	IF Cylinder.List.fbUpCV_FeedInPress1.xError THEN
		Cylinder.List.fbUpCV_FeedInPress1.M_Reset();
	END_IF
	IF Cylinder.List.fbUpCV_FeedInPress2.xError THEN
		Cylinder.List.fbUpCV_FeedInPress2.M_Reset();
	END_IF
	IF Cylinder.List.fbUpCV_DiameterPress.xError THEN
		Cylinder.List.fbUpCV_DiameterPress.M_Reset();
	END_IF
	IF Cylinder.List.fbUpCV_CamaraPress1.xError THEN
		Cylinder.List.fbUpCV_CamaraPress1.M_Reset();
	END_IF
	IF Cylinder.List.fbUpCV_CamaraPress2.xError THEN
		Cylinder.List.fbUpCV_CamaraPress2.M_Reset();
	END_IF
	IF Cylinder.List.fbUpCV_CamaraPress3.xError THEN
		Cylinder.List.fbUpCV_CamaraPress3.M_Reset();
	END_IF
	IF Cylinder.List.fbUpCV_CamaraPress4.xError THEN
		Cylinder.List.fbUpCV_CamaraPress4.M_Reset();
	END_IF
	IF Cylinder.List.fbUpCV_Block1.xError THEN
		Cylinder.List.fbUpCV_Block1.M_Reset();
	END_IF
	IF Cylinder.List.fbUpCV_Block2.xError THEN
		Cylinder.List.fbUpCV_Block2.M_Reset();
	END_IF
	IF Cylinder.List.fbUpCV_Block3.xError THEN
		Cylinder.List.fbUpCV_Block3.M_Reset();
	END_IF
	IF Cylinder.List.fbUpCV_DiameterHoriz.xError THEN
		Cylinder.List.fbUpCV_DiameterHoriz.M_Reset();
	END_IF
	IF Cylinder.List.fbUpCV_DiameterVert.xError THEN
		Cylinder.List.fbUpCV_DiameterVert.M_Reset();
	END_IF
	IF Cylinder.List.fbUpCV_DiameterClamp.xError THEN
		Cylinder.List.fbUpCV_DiameterClamp.M_Reset();
	END_IF
	IF Cylinder.List.fbStackPush.xError THEN
		Cylinder.List.fbStackPush.M_Reset();
	END_IF
	IF Cylinder.List.fbPullOutCV_AsidePress1.xError THEN
		Cylinder.List.fbPullOutCV_AsidePress1.M_Reset();
	END_IF
	IF Cylinder.List.fbPullOutCV_AsidePress2.xError THEN
		Cylinder.List.fbPullOutCV_AsidePress2.M_Reset();
	END_IF
	IF Cylinder.List.fbPullOutCV_AsideBlock.xError THEN
		Cylinder.List.fbPullOutCV_AsideBlock.M_Reset();
	END_IF
	IF Cylinder.List.fbPullOutCV_BsidePress1.xError THEN
		Cylinder.List.fbPullOutCV_BsidePress1.M_Reset();
	END_IF
	IF Cylinder.List.fbPullOutCV_BsidePress2.xError THEN
		Cylinder.List.fbPullOutCV_BsidePress2.M_Reset();
	END_IF
	IF Cylinder.List.fbPullOutCV_BsideBlock.xError THEN
		Cylinder.List.fbPullOutCV_BsideBlock.M_Reset();
	END_IF
	IF Cylinder.List.fbLowCV_Press1.xError THEN
		Cylinder.List.fbLowCV_Press1.M_Reset();
	END_IF
	IF Cylinder.List.fbLowCV_Press2.xError THEN
		Cylinder.List.fbLowCV_Press2.M_Reset();
	END_IF
	IF Cylinder.List.fbLowCV_Press3.xError THEN
		Cylinder.List.fbLowCV_Press3.M_Reset();
	END_IF
	IF Cylinder.List.fbLowCV_Press4.xError THEN
		Cylinder.List.fbLowCV_Press4.M_Reset();
	END_IF
	IF Cylinder.List.fbLowCV_Block1.xError THEN
		Cylinder.List.fbLowCV_Block1.M_Reset();
	END_IF
	IF Cylinder.List.fbLowCV_Block2.xError THEN
		Cylinder.List.fbLowCV_Block2.M_Reset();
	END_IF
	IF Cylinder.List.fbAllocateRobot_LeftVert1.xError THEN
		Cylinder.List.fbAllocateRobot_LeftVert1.M_Reset();
	END_IF
	IF Cylinder.List.fbAllocateRobot_LeftVert2.xError THEN
		Cylinder.List.fbAllocateRobot_LeftVert2.M_Reset();
	END_IF
	IF Cylinder.List.fbAllocateRobot_RightVert1.xError THEN
		Cylinder.List.fbAllocateRobot_RightVert1.M_Reset();
	END_IF
	IF Cylinder.List.fbAllocateRobot_RightVert2.xError THEN
		Cylinder.List.fbAllocateRobot_RightVert2.M_Reset();
	END_IF
	IF Cylinder.List.fbAllocateRobot_LeftClamp1.xError THEN
		Cylinder.List.fbAllocateRobot_LeftClamp1.M_Reset();
	END_IF
	IF Cylinder.List.fbAllocateRobot_LeftClamp2.xError THEN
		Cylinder.List.fbAllocateRobot_LeftClamp2.M_Reset();
	END_IF
	IF Cylinder.List.fbAllocateRobot_RightClamp1.xError THEN
		Cylinder.List.fbAllocateRobot_RightClamp1.M_Reset();
	END_IF
	IF Cylinder.List.fbAllocateRobot_RightClamp2.xError THEN
		Cylinder.List.fbAllocateRobot_RightClamp2.M_Reset();
	END_IF
	IF Cylinder.List.fbRoundBelt_WorkZone_Press.xError THEN
		Cylinder.List.fbRoundBelt_WorkZone_Press.M_Reset();
	END_IF
	IF Cylinder.List.fbRoundBelt_WorkZone_Plug.xError THEN
		Cylinder.List.fbRoundBelt_WorkZone_Plug.M_Reset();
	END_IF
	IF Cylinder.List.fbRoundBelt_ChargeZone_Plug.xError THEN
		Cylinder.List.fbRoundBelt_ChargeZone_Plug.M_Reset();
	END_IF
	IF Cylinder.List.fbRoundBelt_TransmitCVZone_Plug.xError THEN
		Cylinder.List.fbRoundBelt_TransmitCVZone_Plug.M_Reset();
	END_IF
	IF Cylinder.List.fbOutRobot_AsideVert.xError THEN
		Cylinder.List.fbOutRobot_AsideVert.M_Reset();
	END_IF
	IF Cylinder.List.fbOutRobot_BsideVert.xError THEN
		Cylinder.List.fbOutRobot_BsideVert.M_Reset();
	END_IF
	IF Cylinder.List.fbOutRobot_AsideClamp.xError THEN
		Cylinder.List.fbOutRobot_AsideClamp.M_Reset();
	END_IF
	IF Cylinder.List.fbOutRobot_BsideClamp.xError THEN
		Cylinder.List.fbOutRobot_BsideClamp.M_Reset();
	END_IF
	IF Cylinder.List.fbTransmitCV_CamaraHoriz.xError THEN
		Cylinder.List.fbTransmitCV_CamaraHoriz.M_Reset();
	END_IF
	IF Cylinder.List.fbDifferentSizeCV_Press2.xError THEN
		Cylinder.List.fbDifferentSizeCV_Press2.M_Reset();
	END_IF
	IF Cylinder.List.fbDifferentSizeCV_Press1.xError THEN
		Cylinder.List.fbDifferentSizeCV_Press1.M_Reset();
	END_IF
	IF Cylinder.List.fbDifferentSizeCV_Block1.xError THEN
		Cylinder.List.fbDifferentSizeCV_Block1.M_Reset();
	END_IF
	IF Cylinder.List.fbSameSizeCV_Press4.xError THEN
		Cylinder.List.fbSameSizeCV_Press4.M_Reset();
	END_IF
	IF Cylinder.List.fbSameSizeCV_Press3.xError THEN
		Cylinder.List.fbSameSizeCV_Press3.M_Reset();
	END_IF
	IF Cylinder.List.fbSameSizeCV_Press2.xError THEN
		Cylinder.List.fbSameSizeCV_Press2.M_Reset();
	END_IF
	IF Cylinder.List.fbSameSizeCV_Press1.xError THEN
		Cylinder.List.fbSameSizeCV_Press1.M_Reset();
	END_IF
	IF Cylinder.List.fbSameSizeCV_Block2.xError THEN
		Cylinder.List.fbSameSizeCV_Block2.M_Reset();
	END_IF
	IF Cylinder.List.fbSameSizeCV_Block1.xError THEN
		Cylinder.List.fbSameSizeCV_Block1.M_Reset();
	END_IF
	IF Cylinder.List.fbTurntable_Press.xError THEN
		Cylinder.List.fbTurntable_Press.M_Reset();
	END_IF
	{endregion}
	

//////////// Motor
{region Motor}
IF Motor.List.WareHouseCV_01.xError THEN
		Motor.List.WareHouseCV_01.M_Reset();
	END_IF
	IF Motor.List.WareHouseCV_02.xError THEN
		Motor.List.WareHouseCV_02.M_Reset();
	END_IF
	IF Motor.List.WareHouseCV_03.xError THEN
		Motor.List.WareHouseCV_03.M_Reset();
	END_IF
	IF Motor.List.WareHouseCV_04.xError THEN
		Motor.List.WareHouseCV_04.M_Reset();
	END_IF
	IF Motor.List.WareHouseCV_05.xError THEN
		Motor.List.WareHouseCV_05.M_Reset();
	END_IF
	IF Motor.List.WareHouseCV_06.xError THEN
		Motor.List.WareHouseCV_06.M_Reset();
	END_IF
	IF Motor.List.WareHouseCV_07.xError THEN
		Motor.List.WareHouseCV_07.M_Reset();
	END_IF
	IF Motor.List.WareHouseCV_08.xError THEN
		Motor.List.WareHouseCV_08.M_Reset();
	END_IF
	IF Motor.List.WareHouseCV_09.xError THEN
		Motor.List.WareHouseCV_09.M_Reset();
	END_IF
	IF Motor.List.WareHouseCV_10.xError THEN
		Motor.List.WareHouseCV_10.M_Reset();
	END_IF
	IF Motor.List.WareHouseCV_11.xError THEN
		Motor.List.WareHouseCV_11.M_Reset();
	END_IF
	IF Motor.List.WareHouseCV_12.xError THEN
		Motor.List.WareHouseCV_12.M_Reset();
	END_IF
	IF Motor.List.WareHouseCV_13.xError THEN
		Motor.List.WareHouseCV_13.M_Reset();
	END_IF
	IF Motor.List.WareHouseCV_14.xError THEN
		Motor.List.WareHouseCV_14.M_Reset();
	END_IF
	IF Motor.List.WareHouseCV_15.xError THEN
		Motor.List.WareHouseCV_15.M_Reset();
	END_IF
	IF Motor.List.WareHouseCV_16.xError THEN
		Motor.List.WareHouseCV_16.M_Reset();
	END_IF
	IF Motor.List.WareHouseCV_17.xError THEN
		Motor.List.WareHouseCV_17.M_Reset();
	END_IF
	IF Motor.List.WareHouseCV_18.xError THEN
		Motor.List.WareHouseCV_18.M_Reset();
	END_IF
	IF Motor.List.WareHouseCV_19.xError THEN
		Motor.List.WareHouseCV_19.M_Reset();
	END_IF
	IF Motor.List.WareHouseCV_20.xError THEN
		Motor.List.WareHouseCV_20.M_Reset();
	END_IF
	IF Motor.List.UpCV.xError THEN
		Motor.List.UpCV.M_Reset();
	END_IF
	IF Motor.List.LowCV.xError THEN
		Motor.List.LowCV.M_Reset();
	END_IF
	IF Motor.List.PullOutCV_A.xError THEN
		Motor.List.PullOutCV_A.M_Reset();
	END_IF
	IF Motor.List.PullOutCV_B.xError THEN
		Motor.List.PullOutCV_B.M_Reset();
	END_IF
	IF Motor.List.TransmitSameSideCV.xError THEN
		Motor.List.TransmitSameSideCV.M_Reset();
	END_IF
	IF Motor.List.TransmitDifferentSideCV.xError THEN
		Motor.List.TransmitDifferentSideCV.M_Reset();
	END_IF	 
{endregion}
	


ELSIF ResetEdgeDetect.xFallingEdge THEN
	arAxisCtrl_gb[AxisNo.Allocate_X].Admin.ClearError := Machine_Reset;
	arAxisCtrl_gb[AxisNo.Allocate_Y].Admin.ClearError := Machine_Reset;
	arAxisCtrl_gb[AxisNo.OutRobot_X].Admin.ClearError := Machine_Reset;
	arAxisCtrl_gb[AxisNo.OutRobot_Y].Admin.ClearError := Machine_Reset;
	arAxisCtrl_gb[AxisNo.RoundBelt].Admin.ClearError := Machine_Reset;
	arAxisCtrl_gb[AxisNo.TurnTable].Admin.ClearError := Machine_Reset;
	arAxisCtrl_gb[AxisNo.RackMotor].Admin.ClearError := Machine_Reset;
END_IF

Error := xError;
ErrorID := xErrorID;
ErrMsg := xErrorMsg;
END_ACTION

METHOD M_Aborted
VAR
	CylinderIndex :INT;
	MotorIndex : INT;
	ServoIndex : INT;
END_VAR
IF eModeCommand = E_UnitMode.Auto THEN
    GVL_Machine.PackTags[UnitNo.Storage].Command.UnitMode := E_UnitMode.Auto;
    GVL_Machine.PackTags[UnitNo.Allocate].Command.UnitMode := E_UnitMode.Auto;
    GVL_Machine.PackTags[UnitNo.Shipping].Command.UnitMode := E_UnitMode.Auto;
ELSIF eModeCommand = E_UnitMode.Manual THEN
    GVL_Machine.PackTags[UnitNo.Storage].Command.UnitMode := E_UnitMode.Manual;
    GVL_Machine.PackTags[UnitNo.Allocate].Command.UnitMode := E_UnitMode.Manual;
    GVL_Machine.PackTags[UnitNo.Shipping].Command.UnitMode := E_UnitMode.Manual;
END_IF

FOR ServoIndex := 1 TO 7 DO
    arAxisCtrl_gb[ServoIndex].Admin._OpMode.en := ModeAH;
END_FOR

CASE eModeCurrent OF
    E_UnitMode.Manual:
        IF GVL_Machine.PackTags[UnitNo.Allocate].Status.UnitModeCurrent = E_UnitMode.Manual AND
            GVL_Machine.PackTags[UnitNo.Allocate].Status.StateCurrent = ePMLState_Aborted AND
            GVL_Machine.PackTags[UnitNo.Storage].Status.UnitModeCurrent = E_UnitMode.Manual AND
            GVL_Machine.PackTags[UnitNo.Storage].Status.StateCurrent = ePMLState_Aborted AND
            GVL_Machine.PackTags[UnitNo.Shipping].Status.UnitModeCurrent = E_UnitMode.Manual AND
            GVL_Machine.PackTags[UnitNo.Shipping].Status.StateCurrent = ePMLState_Aborted THEN
            IF NOT Error OR Machine_Reset THEN
                M_StateComplete();
            END_IF
        END_IF
    E_UnitMode.Auto:
        IF GVL_Machine.PackTags[UnitNo.Allocate].Status.UnitModeCurrent = E_UnitMode.Auto AND
            GVL_Machine.PackTags[UnitNo.Allocate].Status.StateCurrent = ePMLState_Aborted AND
            GVL_Machine.PackTags[UnitNo.Storage].Status.UnitModeCurrent = E_UnitMode.Auto AND
            GVL_Machine.PackTags[UnitNo.Storage].Status.StateCurrent = ePMLState_Aborted AND
            GVL_Machine.PackTags[UnitNo.Shipping].Status.UnitModeCurrent = E_UnitMode.Auto AND
            GVL_Machine.PackTags[UnitNo.Shipping].Status.StateCurrent = ePMLState_Aborted THEN
            IF NOT Error OR Machine_Reset THEN
                M_StateComplete();
            END_IF
        END_IF
END_CASE
END_METHOD

METHOD M_Aborting
VAR
	CylinderIndex :INT;
	MotorIndex : INT;
	ServoIndex : INT;
END_VAR
CASE eModeCurrent OF
    E_UnitMode.Manual:
        GVL_Machine.PackTags[UnitNo.Allocate].Command.UnitMode := E_UnitMode.Manual;
        GVL_Machine.PackTags[UnitNo.Allocate].Command.CntrlCmd := ePMLCommand_Abort;
        GVL_Machine.PackTags[UnitNo.Storage].Command.UnitMode  := E_UnitMode.Manual;
        GVL_Machine.PackTags[UnitNo.Storage].Command.CntrlCmd  := ePMLCommand_Abort;
        GVL_Machine.PackTags[UnitNo.Shipping].Command.UnitMode := E_UnitMode.Manual;
        GVL_Machine.PackTags[UnitNo.Shipping].Command.CntrlCmd := ePMLCommand_Abort;
		FOR CylinderIndex := 1 TO 53 DO
			Cylinder.arCylinder[CylinderIndex].xEnable := FALSE;
		END_FOR
		FOR MotorIndex := 1 TO 26 DO
			Motor.arMotor[MotorIndex].xEnable := FALSE;
		END_FOR
		TableMove.xExecute := FALSE;
        IF GVL_Machine.PackTags[UnitNo.Allocate].Status.UnitModeCurrent = E_UnitMode.Manual AND
           GVL_Machine.PackTags[UnitNo.Allocate].Status.StateCurrent = ePMLState_Aborting AND
           GVL_Machine.PackTags[UnitNo.Storage].Status.UnitModeCurrent = E_UnitMode.Manual AND
           GVL_Machine.PackTags[UnitNo.Storage].Status.StateCurrent = ePMLState_Aborting AND
           GVL_Machine.PackTags[UnitNo.Shipping].Status.UnitModeCurrent = E_UnitMode.Manual AND
           GVL_Machine.PackTags[UnitNo.Shipping].Status.StateCurrent = ePMLState_Aborting AND NOT
		   TableMove.xError
            THEN
            M_StateComplete();
        END_IF
	E_UnitMode.Auto:
        GVL_Machine.PackTags[UnitNo.Allocate].Command.UnitMode := E_UnitMode.Auto;
        GVL_Machine.PackTags[UnitNo.Allocate].Command.CntrlCmd := ePMLCommand_Abort;
        GVL_Machine.PackTags[UnitNo.Storage].Command.UnitMode  := E_UnitMode.Auto;
        GVL_Machine.PackTags[UnitNo.Storage].Command.CntrlCmd  := ePMLCommand_Abort;
        GVL_Machine.PackTags[UnitNo.Shipping].Command.UnitMode := E_UnitMode.Auto;
        GVL_Machine.PackTags[UnitNo.Shipping].Command.CntrlCmd := ePMLCommand_Abort;
		FOR CylinderIndex := 1 TO 53 DO
			Cylinder.arCylinder[CylinderIndex].xEnable := FALSE;
		END_FOR
		FOR MotorIndex := 1 TO 26 DO
			Motor.arMotor[MotorIndex].xEnable := FALSE;
		END_FOR
		TableMove.xExecute := FALSE;
        IF GVL_Machine.PackTags[UnitNo.Allocate].Status.UnitModeCurrent = E_UnitMode.Auto AND
           GVL_Machine.PackTags[UnitNo.Allocate].Status.StateCurrent = ePMLState_Aborting AND
           GVL_Machine.PackTags[UnitNo.Storage].Status.UnitModeCurrent = E_UnitMode.Auto AND
           GVL_Machine.PackTags[UnitNo.Storage].Status.StateCurrent = ePMLState_Aborting AND
           GVL_Machine.PackTags[UnitNo.Shipping].Status.UnitModeCurrent = E_UnitMode.Auto AND
           GVL_Machine.PackTags[UnitNo.Shipping].Status.StateCurrent = ePMLState_Aborting AND NOT
		   TableMove.xError
            THEN
            M_StateComplete();
        END_IF
END_CASE
FOR ServoIndex:=1 TO 7 DO
	arAxisCtrl_gb[ServoIndex].Admin._OpMode.en := ModeAH;
END_FOR
END_METHOD

METHOD PRIVATE M_Auto_Axes : BOOL
VAR_INPUT
END_VAR

VAR_INST
	AllowAllocateRobotMove : BOOL;
	AllowOutRobotMove : BOOL;
	AllowRoundBeltMove : BOOL;
	AllowTurnTable		:BOOL;
	AllowRackMotor		:BOOL;
END_VAR
// Safe check
AllowAllocateRobotMove := Cylinder.List.fbAllocateRobot_LeftVert1.InRearPosition AND
    Cylinder.List.fbAllocateRobot_LeftVert2.InRearPosition AND
    Cylinder.List.fbAllocateRobot_RightVert1.InRearPosition AND
    Cylinder.List.fbAllocateRobot_RightVert2.InRearPosition;

AllowOutRobotMove := Cylinder.List.fbOutRobot_AsideVert.InRearPosition AND Cylinder.List.fbOutRobot_BsideVert.InRearPosition;
AllowRoundBeltMove := Cylinder.List.fbRoundBelt_ChargeZone_Plug.InRearPosition AND
    Cylinder.List.fbRoundBelt_TransmitCVZone_Plug.InRearPosition AND
    Cylinder.List.fbRoundBelt_WorkZone_Plug.InRearPosition AND
    Cylinder.List.fbRoundBelt_WorkZone_Press.InRearPosition AND
    AllowAllocateRobotMove AND
    AllowOutRobotMove
	AND NOT FanucRobot.List.StorageRobot.BZoneInWork AND NOT FanucRobot.List.StorageRobot.Bzone_AllowWork;;

AllowTurnTable := Cylinder.List.fbTurntable_Press.InRearPosition;
AllowRackMotor := Cylinder.List.fbStackPush.InRearPosition;

// Axis controll
{region "AllocateRobot AxisX"}

IF AllocateManualCommand.AllocatedRobot.AxisX.JOG.MoveFWD AND AllowAllocateRobotMove THEN
    arAxisCtrl_gb[AxisNo.Allocate_X].VelMode.Acc := CurrentData.Axes.Allocate_X.Manual.JogAcceleration;
    arAxisCtrl_gb[AxisNo.Allocate_X].VelMode.Dec := CurrentData.Axes.Allocate_X.Manual.JogDeceleration;
    arAxisCtrl_gb[AxisNo.Allocate_X].VelMode.Jerk := CurrentData.Axes.Allocate_X.Manual.JogJerk;
    arAxisCtrl_gb[AxisNo.Allocate_X].VelMode.Velocity := CurrentData.Axes.Allocate_X.Manual.JogVelocity;
    arAxisCtrl_gb[AxisNo.Allocate_X].Admin._OpMode.en := E_AXIS_MODE.ModeVel;
ELSIF AllocateManualCommand.AllocatedRobot.AxisX.JOG.MoveBWD AND AllowAllocateRobotMove THEN
    arAxisCtrl_gb[AxisNo.Allocate_X].VelMode.Acc := CurrentData.Axes.Allocate_X.Manual.JogAcceleration;
    arAxisCtrl_gb[AxisNo.Allocate_X].VelMode.Dec := CurrentData.Axes.Allocate_X.Manual.JogDeceleration;
    arAxisCtrl_gb[AxisNo.Allocate_X].VelMode.Jerk := CurrentData.Axes.Allocate_X.Manual.JogJerk;
    arAxisCtrl_gb[AxisNo.Allocate_X].VelMode.Velocity := CurrentData.Axes.Allocate_X.Manual.JogVelocity * -1;
    arAxisCtrl_gb[AxisNo.Allocate_X].Admin._OpMode.en := E_AXIS_MODE.ModeVel;
ELSIF AllocateManualCommand.AllocatedRobot.AxisX.PTP.Enable AND AllowAllocateRobotMove THEN
    arAxisCtrl_gb[AxisNo.Allocate_X].PosMode.Acc := CurrentData.Axes.Allocate_X.Manual.PtpAcceleration;
    arAxisCtrl_gb[AxisNo.Allocate_X].PosMode.Dec := CurrentData.Axes.Allocate_X.Manual.PtpDeceleration;
    arAxisCtrl_gb[AxisNo.Allocate_X].PosMode.Jerk := CurrentData.Axes.Allocate_X.Manual.PtpJerk;
    arAxisCtrl_gb[AxisNo.Allocate_X].PosMode.Velocity := CurrentData.Axes.Allocate_X.Manual.PtpVelocity;
    arAxisCtrl_gb[AxisNo.Allocate_X].PosMode.Position := CurrentData.Axes.Allocate_X.Manual.PtpPosition;
    arAxisCtrl_gb[AxisNo.Allocate_X].Admin._OpMode.en := ModePosAbs;
ELSIF (AllocateManualCommand.AllocatedRobot.AxisX.Homing.Execute OR  fbAllocateArea.fbAllocateHome.AxisHomingRequest)  AND AllowAllocateRobotMove THEN
    arAxisCtrl_gb[AxisNo.Allocate_X].SetupMode.eHomingMode := E_HomingMode._17_Neg_LimitOutterRight;
    arAxisCtrl_gb[AxisNo.Allocate_X].SetupMode.FastVelo := CurrentData.Axes.Allocate_X.Homing.FastVelo;
    arAxisCtrl_gb[AxisNo.Allocate_X].SetupMode.SlowVelo := CurrentData.Axes.Allocate_X.Homing.SlowVelo;
    arAxisCtrl_gb[AxisNo.Allocate_X].SetupMode.lrOffset := CurrentData.Axes.Allocate_X.Homing.Offset;
    arAxisCtrl_gb[AxisNo.Allocate_X].SetupMode.lrSetPosition := CurrentData.Axes.Allocate_X.Homing.SetAbsolutePosition;
    arAxisCtrl_gb[AxisNo.Allocate_X].SetupMode.stPosBiasParameter.bSetPostionBias := TRUE;
    arAxisCtrl_gb[AxisNo.Allocate_X].Admin._OpMode.en := ModeHoming;
ELSIF TableMove.xBusy AND AllowAllocateRobotMove THEN
    arAxisCtrl_gb[AxisNo.Allocate_X].Admin._OpMode.en := ModePosAbs;
ELSIF (fbAllocateArea.fb_AllocateBatchMode.Busy OR fbAllocateArea.fb_AllocateBatchMode_Reverse.Busy ) AND AllowAllocateRobotMove THEN
    arAxisCtrl_gb[AxisNo.Allocate_X].Admin._OpMode.en := ModePosAbs;
		 
ELSE
    arAxisCtrl_gb[AxisNo.Allocate_X].Admin.StopDeceleration := 1000;
    arAxisCtrl_gb[AxisNo.Allocate_X].Admin._OpMode.en := E_AXIS_MODE.ModeAH;
		 
END_IF
{endregion}

{region "AllocateRobot AxisY"}
IF AllocateManualCommand.AllocatedRobot.AxisY.JOG.MoveFWD AND AllowAllocateRobotMove THEN
    arAxisCtrl_gb[AxisNo.Allocate_Y].VelMode.Acc := CurrentData.Axes.Allocate_Y.Manual.JogAcceleration;
    arAxisCtrl_gb[AxisNo.Allocate_Y].VelMode.Dec := CurrentData.Axes.Allocate_Y.Manual.JogDeceleration;
    arAxisCtrl_gb[AxisNo.Allocate_Y].VelMode.Jerk := CurrentData.Axes.Allocate_Y.Manual.JogJerk;
    arAxisCtrl_gb[AxisNo.Allocate_Y].VelMode.Velocity := CurrentData.Axes.Allocate_Y.Manual.JogVelocity;
    arAxisCtrl_gb[AxisNo.Allocate_Y].Admin._OpMode.en := E_AXIS_MODE.ModeVel;
ELSIF AllocateManualCommand.AllocatedRobot.AxisY.JOG.MoveBWD AND AllowAllocateRobotMove THEN
    arAxisCtrl_gb[AxisNo.Allocate_Y].VelMode.Acc := CurrentData.Axes.Allocate_Y.Manual.JogAcceleration;
    arAxisCtrl_gb[AxisNo.Allocate_Y].VelMode.Dec := CurrentData.Axes.Allocate_Y.Manual.JogDeceleration;
    arAxisCtrl_gb[AxisNo.Allocate_Y].VelMode.Jerk := CurrentData.Axes.Allocate_Y.Manual.JogJerk;
    arAxisCtrl_gb[AxisNo.Allocate_Y].VelMode.Velocity := CurrentData.Axes.Allocate_Y.Manual.JogVelocity * -1;
    arAxisCtrl_gb[AxisNo.Allocate_Y].Admin._OpMode.en := E_AXIS_MODE.ModeVel;
ELSIF AllocateManualCommand.AllocatedRobot.AxisY.PTP.Enable AND AllowAllocateRobotMove THEN
    arAxisCtrl_gb[AxisNo.Allocate_Y].PosMode.Acc := CurrentData.Axes.Allocate_Y.Manual.PtpAcceleration;
    arAxisCtrl_gb[AxisNo.Allocate_Y].PosMode.Dec := CurrentData.Axes.Allocate_Y.Manual.PtpDeceleration;
    arAxisCtrl_gb[AxisNo.Allocate_Y].PosMode.Jerk := CurrentData.Axes.Allocate_Y.Manual.PtpJerk;
    arAxisCtrl_gb[AxisNo.Allocate_Y].PosMode.Velocity := CurrentData.Axes.Allocate_Y.Manual.PtpVelocity;
    arAxisCtrl_gb[AxisNo.Allocate_Y].PosMode.Position := CurrentData.Axes.Allocate_Y.Manual.PtpPosition;
    arAxisCtrl_gb[AxisNo.Allocate_Y].Admin._OpMode.en := ModePosAbs;
//ELSIF( AllocateManualCommand.AllocatedRobot.AxisY.Homing.Execute OR  fbAllocateArea.fbAllocateHome.AxisHomingRequest ) AND AllowAllocateRobotMove THEN
//    arAxisCtrl_gb[AxisNo.Allocate_Y].SetupMode.eHomingMode := E_HomingMode._36_MoveToAbsHomePoint;
//    arAxisCtrl_gb[AxisNo.Allocate_Y].SetupMode.FastVelo := CurrentData.Axes.Allocate_Y.Homing.FastVelo;
//    arAxisCtrl_gb[AxisNo.Allocate_Y].SetupMode.SlowVelo := CurrentData.Axes.Allocate_Y.Homing.SlowVelo;
//    arAxisCtrl_gb[AxisNo.Allocate_Y].SetupMode.lrOffset := CurrentData.Axes.Allocate_Y.Homing.Offset;
//    arAxisCtrl_gb[AxisNo.Allocate_Y].SetupMode.lrSetPosition := CurrentData.Axes.Allocate_Y.Homing.SetAbsolutePosition;
//    arAxisCtrl_gb[AxisNo.Allocate_Y].SetupMode.stPosBiasParameter.bSetPostionBias := FALSE;
//    arAxisCtrl_gb[AxisNo.Allocate_Y].Admin._OpMode.en := ModeHoming;
ELSIF( AllocateManualCommand.AllocatedRobot.AxisY.Homing.Execute OR  fbAllocateArea.fbAllocateHome.AxisHomingRequest ) AND AllowAllocateRobotMove THEN
    arAxisCtrl_gb[AxisNo.Allocate_Y].PosMode.Acc := CurrentData.Axes.Allocate_Y.Homing.FastVelo.Acc;
    arAxisCtrl_gb[AxisNo.Allocate_Y].PosMode.Dec := CurrentData.Axes.Allocate_Y.Homing.FastVelo.Dec;
    arAxisCtrl_gb[AxisNo.Allocate_Y].PosMode.Jerk := CurrentData.Axes.Allocate_Y.Homing.FastVelo.Jerk;
    arAxisCtrl_gb[AxisNo.Allocate_Y].PosMode.Velocity := CurrentData.Axes.Allocate_Y.Homing.FastVelo.Velocity;
    arAxisCtrl_gb[AxisNo.Allocate_Y].PosMode.Position := CurrentData.Axes.Allocate_Y.Homing.Offset;
    arAxisCtrl_gb[AxisNo.Allocate_Y].Admin._OpMode.en := ModePosAbs;
		 
    IF arAxisStatus_gb[AxisNo.Allocate_Y].Admin._OpModeAck = ModePosAbs AND arAxisStatus_gb[AxisNo.Allocate_Y].Admin.CmdDone THEN
        GVL_Machine.AllocatYAxisHome := TRUE;
    END_IF
ELSIF TableMove.xBusy AND AllowAllocateRobotMove THEN
    arAxisCtrl_gb[AxisNo.Allocate_Y].Admin._OpMode.en := ModePosAbs;
ELSIF (fbAllocateArea.fb_AllocateBatchMode.Busy OR fbAllocateArea.fb_AllocateBatchMode_Reverse.Busy) AND AllowAllocateRobotMove THEN
    arAxisCtrl_gb[AxisNo.Allocate_Y].Admin._OpMode.en := ModePosAbs;
ELSE
    arAxisCtrl_gb[AxisNo.Allocate_Y].Admin.StopDeceleration := 1000;
    arAxisCtrl_gb[AxisNo.Allocate_Y].Admin._OpMode.en := E_AXIS_MODE.ModeAH;
END_IF

{EndRegion}

{region "OutRobot AxisX"}
IF AllocateManualCommand.OutRobot.AxisX.JOG.MoveFWD AND AllowOutRobotMove THEN
    arAxisCtrl_gb[AxisNo.OutRobot_X].VelMode.Acc := CurrentData.Axes.OutRobot_X.Manual.JogAcceleration;
    arAxisCtrl_gb[AxisNo.OutRobot_X].VelMode.Dec := CurrentData.Axes.OutRobot_X.Manual.JogDeceleration;
    arAxisCtrl_gb[AxisNo.OutRobot_X].VelMode.Jerk := CurrentData.Axes.OutRobot_X.Manual.JogJerk;
    arAxisCtrl_gb[AxisNo.OutRobot_X].VelMode.Velocity := CurrentData.Axes.OutRobot_X.Manual.JogVelocity;
    arAxisCtrl_gb[AxisNo.OutRobot_X].Admin._OpMode.en := E_AXIS_MODE.ModeVel;
ELSIF AllocateManualCommand.OutRobot.AxisX.JOG.MoveBWD AND AllowOutRobotMove THEN
    arAxisCtrl_gb[AxisNo.OutRobot_X].VelMode.Acc := CurrentData.Axes.OutRobot_X.Manual.JogAcceleration;
    arAxisCtrl_gb[AxisNo.OutRobot_X].VelMode.Dec := CurrentData.Axes.OutRobot_X.Manual.JogDeceleration;
    arAxisCtrl_gb[AxisNo.OutRobot_X].VelMode.Jerk := CurrentData.Axes.OutRobot_X.Manual.JogJerk;
    arAxisCtrl_gb[AxisNo.OutRobot_X].VelMode.Velocity := CurrentData.Axes.OutRobot_X.Manual.JogVelocity * -1;
    arAxisCtrl_gb[AxisNo.OutRobot_X].Admin._OpMode.en := E_AXIS_MODE.ModeVel;
ELSIF AllocateManualCommand.OutRobot.AxisX.PTP.Enable AND AllowOutRobotMove THEN
    arAxisCtrl_gb[AxisNo.OutRobot_X].PosMode.Acc := CurrentData.Axes.OutRobot_X.Manual.PtpAcceleration;
    arAxisCtrl_gb[AxisNo.OutRobot_X].PosMode.Dec := CurrentData.Axes.OutRobot_X.Manual.PtpDeceleration;
    arAxisCtrl_gb[AxisNo.OutRobot_X].PosMode.Jerk := CurrentData.Axes.OutRobot_X.Manual.PtpJerk;
    arAxisCtrl_gb[AxisNo.OutRobot_X].PosMode.Velocity := CurrentData.Axes.OutRobot_X.Manual.PtpVelocity;
    arAxisCtrl_gb[AxisNo.OutRobot_X].PosMode.Position := CurrentData.Axes.OutRobot_X.Manual.PtpPosition;
    arAxisCtrl_gb[AxisNo.OutRobot_X].Admin._OpMode.en := ModePosAbs;
ELSIF (AllocateManualCommand.OutRobot.AxisX.Homing.Execute OR  fbAllocateArea.fbAllocateHome.AxisHomingRequest ) AND AllowOutRobotMove THEN
    arAxisCtrl_gb[AxisNo.OutRobot_X].SetupMode.eHomingMode := E_HomingMode._28_Neg_HomeInnerRight_withLimit;
    arAxisCtrl_gb[AxisNo.OutRobot_X].SetupMode.FastVelo := CurrentData.Axes.OutRobot_X.Homing.FastVelo;
    arAxisCtrl_gb[AxisNo.OutRobot_X].SetupMode.SlowVelo := CurrentData.Axes.OutRobot_X.Homing.SlowVelo;
    arAxisCtrl_gb[AxisNo.OutRobot_X].SetupMode.lrOffset := CurrentData.Axes.OutRobot_X.Homing.Offset;
    arAxisCtrl_gb[AxisNo.OutRobot_X].SetupMode.lrSetPosition := CurrentData.Axes.OutRobot_X.Homing.SetAbsolutePosition;
    arAxisCtrl_gb[AxisNo.OutRobot_X].SetupMode.stPosBiasParameter.bSetPostionBias := TRUE;
    arAxisCtrl_gb[AxisNo.OutRobot_X].Admin._OpMode.en := ModeHoming;
ELSIF (TableMove.xBusy OR AllocateService.AutoMode_BoxMoveReverse.HandShake.Busy 
	  OR AllocateService.AutoMode_EmptyBoxMove.HandShake.Busy 
	  OR AllocateService.AutoMode_RareBoxMove.HandShake.Busy) AND AllowOutRobotMove THEN
	arAxisCtrl_gb[AxisNo.OutRobot_X].PosMode.Acc := CurrentData.Axes.OutRobot_X.HalfAuto.Acceleration;
    arAxisCtrl_gb[AxisNo.OutRobot_X].PosMode.Dec := CurrentData.Axes.OutRobot_X.HalfAuto.Deceleration;
    arAxisCtrl_gb[AxisNo.OutRobot_X].PosMode.Jerk := CurrentData.Axes.OutRobot_X.HalfAuto.Jerk;
    arAxisCtrl_gb[AxisNo.OutRobot_X].PosMode.Velocity := CurrentData.Axes.OutRobot_X.HalfAuto.Velocity;		   
    arAxisCtrl_gb[AxisNo.OutRobot_X].Admin._OpMode.en := ModePosAbs;
ELSE
    arAxisCtrl_gb[AxisNo.OutRobot_X].Admin.StopDeceleration := 1000;
    arAxisCtrl_gb[AxisNo.OutRobot_X].Admin._OpMode.en := E_AXIS_MODE.ModeAH;
END_IF

{Endregion}

{region "OutRobot AxisY"}
IF AllocateManualCommand.OutRobot.AxisY.JOG.MoveFWD AND AllowOutRobotMove THEN
    arAxisCtrl_gb[AxisNo.OutRobot_Y].VelMode.Acc := CurrentData.Axes.OutRobot_Y.Manual.JogAcceleration;
    arAxisCtrl_gb[AxisNo.OutRobot_Y].VelMode.Dec := CurrentData.Axes.OutRobot_Y.Manual.JogDeceleration;
    arAxisCtrl_gb[AxisNo.OutRobot_Y].VelMode.Jerk := CurrentData.Axes.OutRobot_Y.Manual.JogJerk;
    arAxisCtrl_gb[AxisNo.OutRobot_Y].VelMode.Velocity := CurrentData.Axes.OutRobot_Y.Manual.JogVelocity;
    arAxisCtrl_gb[AxisNo.OutRobot_Y].Admin._OpMode.en := E_AXIS_MODE.ModeVel;
ELSIF AllocateManualCommand.OutRobot.AxisY.JOG.MoveBWD AND AllowOutRobotMove THEN
    arAxisCtrl_gb[AxisNo.OutRobot_Y].VelMode.Acc := CurrentData.Axes.OutRobot_Y.Manual.JogAcceleration;
    arAxisCtrl_gb[AxisNo.OutRobot_Y].VelMode.Dec := CurrentData.Axes.OutRobot_Y.Manual.JogDeceleration;
    arAxisCtrl_gb[AxisNo.OutRobot_Y].VelMode.Jerk := CurrentData.Axes.OutRobot_Y.Manual.JogJerk;
    arAxisCtrl_gb[AxisNo.OutRobot_Y].VelMode.Velocity := CurrentData.Axes.OutRobot_Y.Manual.JogVelocity * -1;
    arAxisCtrl_gb[AxisNo.OutRobot_Y].Admin._OpMode.en := E_AXIS_MODE.ModeVel;
ELSIF AllocateManualCommand.OutRobot.AxisY.PTP.Enable AND AllowOutRobotMove THEN
    arAxisCtrl_gb[AxisNo.OutRobot_Y].PosMode.Acc := CurrentData.Axes.OutRobot_Y.Manual.PtpAcceleration;
    arAxisCtrl_gb[AxisNo.OutRobot_Y].PosMode.Dec := CurrentData.Axes.OutRobot_Y.Manual.PtpDeceleration;
    arAxisCtrl_gb[AxisNo.OutRobot_Y].PosMode.Jerk := CurrentData.Axes.OutRobot_Y.Manual.PtpJerk;
    arAxisCtrl_gb[AxisNo.OutRobot_Y].PosMode.Velocity := CurrentData.Axes.OutRobot_Y.Manual.PtpVelocity;
    arAxisCtrl_gb[AxisNo.OutRobot_Y].PosMode.Position := CurrentData.Axes.OutRobot_Y.Manual.PtpPosition;
    arAxisCtrl_gb[AxisNo.OutRobot_Y].Admin._OpMode.en := ModePosAbs;
ELSIF (AllocateManualCommand.OutRobot.AxisY.Homing.Execute OR  fbAllocateArea.fbAllocateHome.AxisHomingRequest) AND AllowOutRobotMove THEN
    arAxisCtrl_gb[AxisNo.OutRobot_Y].SetupMode.eHomingMode := E_HomingMode._28_Neg_HomeInnerRight_withLimit;
    arAxisCtrl_gb[AxisNo.OutRobot_Y].SetupMode.FastVelo := CurrentData.Axes.OutRobot_Y.Homing.FastVelo;
    arAxisCtrl_gb[AxisNo.OutRobot_Y].SetupMode.SlowVelo := CurrentData.Axes.OutRobot_Y.Homing.SlowVelo;
    arAxisCtrl_gb[AxisNo.OutRobot_Y].SetupMode.lrOffset := CurrentData.Axes.OutRobot_Y.Homing.Offset;
    arAxisCtrl_gb[AxisNo.OutRobot_Y].SetupMode.lrSetPosition := CurrentData.Axes.OutRobot_Y.Homing.SetAbsolutePosition;
    arAxisCtrl_gb[AxisNo.OutRobot_Y].SetupMode.stPosBiasParameter.bSetPostionBias := TRUE;
    arAxisCtrl_gb[AxisNo.OutRobot_Y].Admin._OpMode.en := ModeHoming;
ELSIF (TableMove.xBusy OR AllocateService.AutoMode_BoxMoveReverse.HandShake.Busy 
	  OR AllocateService.AutoMode_EmptyBoxMove.HandShake.Busy 
	  OR AllocateService.AutoMode_RareBoxMove.HandShake.Busy)AND AllowOutRobotMove THEN
	arAxisCtrl_gb[AxisNo.OutRobot_Y].PosMode.Acc := CurrentData.Axes.OutRobot_Y.HalfAuto.Acceleration;
    arAxisCtrl_gb[AxisNo.OutRobot_Y].PosMode.Dec := CurrentData.Axes.OutRobot_Y.HalfAuto.Deceleration;
    arAxisCtrl_gb[AxisNo.OutRobot_Y].PosMode.Jerk := CurrentData.Axes.OutRobot_Y.HalfAuto.Jerk;
    arAxisCtrl_gb[AxisNo.OutRobot_Y].PosMode.Velocity := CurrentData.Axes.OutRobot_Y.HalfAuto.Velocity;		   
    arAxisCtrl_gb[AxisNo.OutRobot_Y].Admin._OpMode.en := ModePosAbs;
ELSE
    arAxisCtrl_gb[AxisNo.OutRobot_Y].Admin.StopDeceleration := 1000;
    arAxisCtrl_gb[AxisNo.OutRobot_Y].Admin._OpMode.en := E_AXIS_MODE.ModeAH;
END_IF

{Endregion}

{region "RoundBelt Axis"}
IF AllocateManualCommand.RoundBelt.Axis.JOG.MoveFWD AND AllowRoundBeltMove THEN
    arAxisCtrl_gb[AxisNo.RoundBelt].VelMode.Acc := CurrentData.Axes.RoundBelt.Manual.JogAcceleration;
    arAxisCtrl_gb[AxisNo.RoundBelt].VelMode.Dec := CurrentData.Axes.RoundBelt.Manual.JogDeceleration;
    arAxisCtrl_gb[AxisNo.RoundBelt].VelMode.Jerk := CurrentData.Axes.RoundBelt.Manual.JogJerk;
    arAxisCtrl_gb[AxisNo.RoundBelt].VelMode.Velocity := CurrentData.Axes.RoundBelt.Manual.JogVelocity;
    arAxisCtrl_gb[AxisNo.RoundBelt].Admin._OpMode.en := E_AXIS_MODE.ModeVel;
ELSIF AllocateManualCommand.RoundBelt.Axis.JOG.MoveBWD AND AllowRoundBeltMove THEN
    arAxisCtrl_gb[AxisNo.RoundBelt].VelMode.Acc := CurrentData.Axes.RoundBelt.Manual.JogAcceleration;
    arAxisCtrl_gb[AxisNo.RoundBelt].VelMode.Dec := CurrentData.Axes.RoundBelt.Manual.JogDeceleration;
    arAxisCtrl_gb[AxisNo.RoundBelt].VelMode.Jerk := CurrentData.Axes.RoundBelt.Manual.JogJerk;
    arAxisCtrl_gb[AxisNo.RoundBelt].VelMode.Velocity := CurrentData.Axes.RoundBelt.Manual.JogVelocity * -1;
    arAxisCtrl_gb[AxisNo.RoundBelt].Admin._OpMode.en := E_AXIS_MODE.ModeVel;
ELSIF AllocateManualCommand.RoundBelt.Axis.PTP.Enable AND AllowRoundBeltMove THEN
    arAxisCtrl_gb[AxisNo.RoundBelt].PosMode.Acc := CurrentData.Axes.RoundBelt.Manual.PtpAcceleration;
    arAxisCtrl_gb[AxisNo.RoundBelt].PosMode.Dec := CurrentData.Axes.RoundBelt.Manual.PtpDeceleration;
    arAxisCtrl_gb[AxisNo.RoundBelt].PosMode.Jerk := CurrentData.Axes.RoundBelt.Manual.PtpJerk;
    arAxisCtrl_gb[AxisNo.RoundBelt].PosMode.Velocity := CurrentData.Axes.RoundBelt.Manual.PtpVelocity;
    arAxisCtrl_gb[AxisNo.RoundBelt].PosMode.Position := CurrentData.Axes.RoundBelt.Manual.PtpPosition;
    arAxisCtrl_gb[AxisNo.RoundBelt].Admin._OpMode.en := ModePosAbs;
ELSIF (AllocateManualCommand.RoundBelt.Axis.Homing.Execute OR  fbAllocateArea.fbAllocateHome.AxisHomingRequest ) AND AllowRoundBeltMove THEN
    arAxisCtrl_gb[AxisNo.RoundBelt].SetupMode.eHomingMode := E_HomingMode._20_Pos_HomeInnerLeft;
    arAxisCtrl_gb[AxisNo.RoundBelt].SetupMode.FastVelo := CurrentData.Axes.RoundBelt.Homing.FastVelo;
    arAxisCtrl_gb[AxisNo.RoundBelt].SetupMode.SlowVelo := CurrentData.Axes.RoundBelt.Homing.SlowVelo;
    arAxisCtrl_gb[AxisNo.RoundBelt].SetupMode.lrOffset := CurrentData.Axes.RoundBelt.Homing.Offset;
    arAxisCtrl_gb[AxisNo.RoundBelt].SetupMode.lrSetPosition := CurrentData.Axes.RoundBelt.Homing.SetAbsolutePosition;
    arAxisCtrl_gb[AxisNo.RoundBelt].SetupMode.stPosBiasParameter.bSetPostionBias := TRUE;
    arAxisCtrl_gb[AxisNo.RoundBelt].Admin._OpMode.en := ModeHoming;
ELSIF TableMove.xBusy AND AllowRoundBeltMove THEN
    arAxisCtrl_gb[AxisNo.RoundBelt].Admin._OpMode.en := ModePosAbs;
ELSIF AllocateService.AllocateCircleMove.HandShake.Busy AND AllowRoundBeltMove THEN
    arAxisCtrl_gb[AxisNo.RoundBelt].PosMode.Acc := CurrentData.Axes.RoundBelt.HalfAuto.Acceleration;
    arAxisCtrl_gb[AxisNo.RoundBelt].PosMode.Dec := CurrentData.Axes.RoundBelt.HalfAuto.Deceleration;
    arAxisCtrl_gb[AxisNo.RoundBelt].PosMode.Jerk := CurrentData.Axes.RoundBelt.HalfAuto.Jerk;
    arAxisCtrl_gb[AxisNo.RoundBelt].PosMode.Velocity := CurrentData.Axes.RoundBelt.HalfAuto.Velocity;
    arAxisCtrl_gb[AxisNo.RoundBelt].Admin._OpMode.en := ModePosAbs;
ELSIF (AllocateService.AutoMode_AllocateBatchMode.HandShake.Busy OR 
StorageService.AutoMode_ReloadRoundBeltBoxWithRobot.Status.Busy OR 
AllocateService.AutoMode_AllocateBatchMode_Reverse.HandShake.Busy) AND 
AllowRoundBeltMove THEN
    arAxisCtrl_gb[AxisNo.RoundBelt].PosMode.Acc := CurrentData.Axes.RoundBelt.HalfAuto.Acceleration;
    arAxisCtrl_gb[AxisNo.RoundBelt].PosMode.Dec := CurrentData.Axes.RoundBelt.HalfAuto.Deceleration;
    arAxisCtrl_gb[AxisNo.RoundBelt].PosMode.Jerk := CurrentData.Axes.RoundBelt.HalfAuto.Jerk;
    arAxisCtrl_gb[AxisNo.RoundBelt].PosMode.Velocity := CurrentData.Axes.RoundBelt.HalfAuto.Velocity;
    arAxisCtrl_gb[AxisNo.RoundBelt].Admin._OpMode.en := ModePosAbs;
//AutoMode Action
ELSIF (AllocateService.AutoMode_AllocateCircleMove.HandShake.Busy OR 
fbAllocateArea.RoundBeltMoveJob_Status.Busy)AND 
AllowRoundBeltMove THEN
    arAxisCtrl_gb[AxisNo.RoundBelt].PosMode.Acc := CurrentData.Axes.RoundBelt.Auto.Acceleration;
    arAxisCtrl_gb[AxisNo.RoundBelt].PosMode.Dec := CurrentData.Axes.RoundBelt.Auto.Deceleration;
    arAxisCtrl_gb[AxisNo.RoundBelt].PosMode.Jerk := CurrentData.Axes.RoundBelt.Auto.Jerk;
    arAxisCtrl_gb[AxisNo.RoundBelt].PosMode.Velocity := CurrentData.Axes.RoundBelt.Auto.Velocity;
    arAxisCtrl_gb[AxisNo.RoundBelt].Admin._OpMode.en := ModePosAbs;
ELSE
    arAxisCtrl_gb[AxisNo.RoundBelt].Admin.StopDeceleration := 1000;
    arAxisCtrl_gb[AxisNo.RoundBelt].Admin._OpMode.en := E_AXIS_MODE.ModeAH;
END_IF

{endregion}

{region "TurnTable Axis"}
IF AllocateManualCommand.TurnTable.Axis.JOG.MoveFWD AND AllowTurnTable THEN
    arAxisCtrl_gb[AxisNo.TurnTable].VelMode.Acc := CurrentData.Axes.TurnTable.Manual.JogAcceleration;
    arAxisCtrl_gb[AxisNo.TurnTable].VelMode.Dec := CurrentData.Axes.TurnTable.Manual.JogDeceleration;
    arAxisCtrl_gb[AxisNo.TurnTable].VelMode.Jerk := CurrentData.Axes.TurnTable.Manual.JogJerk;
    arAxisCtrl_gb[AxisNo.TurnTable].VelMode.Velocity := CurrentData.Axes.TurnTable.Manual.JogVelocity;
    arAxisCtrl_gb[AxisNo.TurnTable].Admin._OpMode.en := E_AXIS_MODE.ModeVel;
ELSIF AllocateManualCommand.TurnTable.Axis.JOG.MoveBWD THEN
    arAxisCtrl_gb[AxisNo.TurnTable].VelMode.Acc := CurrentData.Axes.TurnTable.Manual.JogAcceleration;
    arAxisCtrl_gb[AxisNo.TurnTable].VelMode.Dec := CurrentData.Axes.TurnTable.Manual.JogDeceleration;
    arAxisCtrl_gb[AxisNo.TurnTable].VelMode.Jerk := CurrentData.Axes.TurnTable.Manual.JogJerk;
    arAxisCtrl_gb[AxisNo.TurnTable].VelMode.Velocity := CurrentData.Axes.TurnTable.Manual.JogVelocity * -1;
    arAxisCtrl_gb[AxisNo.TurnTable].Admin._OpMode.en := E_AXIS_MODE.ModeVel;
ELSIF AllocateManualCommand.TurnTable.Axis.PTP.Enable THEN
    arAxisCtrl_gb[AxisNo.TurnTable].PosMode.Acc := CurrentData.Axes.TurnTable.Manual.PtpAcceleration;
    arAxisCtrl_gb[AxisNo.TurnTable].PosMode.Dec := CurrentData.Axes.TurnTable.Manual.PtpDeceleration;
    arAxisCtrl_gb[AxisNo.TurnTable].PosMode.Jerk := CurrentData.Axes.TurnTable.Manual.PtpJerk;
    arAxisCtrl_gb[AxisNo.TurnTable].PosMode.Velocity := CurrentData.Axes.TurnTable.Manual.PtpVelocity;
    arAxisCtrl_gb[AxisNo.TurnTable].PosMode.Position := CurrentData.Axes.TurnTable.Manual.PtpPosition;
    arAxisCtrl_gb[AxisNo.TurnTable].Admin._OpMode.en := ModePosAbs;
ELSIF (AllocateManualCommand.TurnTable.Axis.Homing.Execute OR  fbAllocateArea.fbAllocateHome.AxisHomingRequest) AND  AllowTurnTable THEN
    arAxisCtrl_gb[AxisNo.TurnTable].SetupMode.eHomingMode := E_HomingMode._22_Neg_HomeInnerRight;
    arAxisCtrl_gb[AxisNo.TurnTable].SetupMode.FastVelo := CurrentData.Axes.TurnTable.Homing.FastVelo;
    arAxisCtrl_gb[AxisNo.TurnTable].SetupMode.SlowVelo := CurrentData.Axes.TurnTable.Homing.SlowVelo;
    arAxisCtrl_gb[AxisNo.TurnTable].SetupMode.lrOffset := CurrentData.Axes.TurnTable.Homing.Offset;
    arAxisCtrl_gb[AxisNo.TurnTable].SetupMode.lrSetPosition := CurrentData.Axes.TurnTable.Homing.SetAbsolutePosition;
    arAxisCtrl_gb[AxisNo.TurnTable].SetupMode.stPosBiasParameter.bSetPostionBias := TRUE;
    arAxisCtrl_gb[AxisNo.TurnTable].Admin._OpMode.en := ModeHoming;
ELSIF TableMove.xBusy AND AllowTurnTable THEN
    arAxisCtrl_gb[AxisNo.TurnTable].Admin._OpMode.en := ModePosAbs;
ELSIF (AllocateService.TurnTableMove.HandShake.Busy ) AND AllowTurnTable THEN
    arAxisCtrl_gb[AxisNo.TurnTable].PosMode.Acc := CurrentData.Axes.TurnTable.HalfAuto.Acceleration;
    arAxisCtrl_gb[AxisNo.TurnTable].PosMode.Dec := CurrentData.Axes.TurnTable.HalfAuto.Deceleration;
    arAxisCtrl_gb[AxisNo.TurnTable].PosMode.Jerk := CurrentData.Axes.TurnTable.HalfAuto.Jerk;
    arAxisCtrl_gb[AxisNo.TurnTable].PosMode.Velocity := CurrentData.Axes.TurnTable.HalfAuto.Velocity;
    arAxisCtrl_gb[AxisNo.TurnTable].Admin._OpMode.en := ModePosAbs;
ELSIF AllocateService.AutoMode_TurnTableMove.HandShake.Busy AND AllowTurnTable THEN
    arAxisCtrl_gb[AxisNo.TurnTable].PosMode.Acc := CurrentData.Axes.TurnTable.Auto.Acceleration;
    arAxisCtrl_gb[AxisNo.TurnTable].PosMode.Dec := CurrentData.Axes.TurnTable.Auto.Deceleration;
    arAxisCtrl_gb[AxisNo.TurnTable].PosMode.Jerk := CurrentData.Axes.TurnTable.Auto.Jerk;
    arAxisCtrl_gb[AxisNo.TurnTable].PosMode.Velocity := CurrentData.Axes.TurnTable.Auto.Velocity;
    arAxisCtrl_gb[AxisNo.TurnTable].Admin._OpMode.en := ModePosAbs;
ELSE
    arAxisCtrl_gb[AxisNo.TurnTable].Admin.StopDeceleration := 1000;
    arAxisCtrl_gb[AxisNo.TurnTable].Admin._OpMode.en := E_AXIS_MODE.ModeAH;
END_IF

{endregion}

{region "Rack motor Axis"}
IF StorageManualCommand.RackMotor.Axis.JOG.MoveFWD AND AllowRackMotor THEN
    arAxisCtrl_gb[AxisNo.RackMotor].VelMode.Acc := CurrentData.Axes.RackMotor.Manual.JogAcceleration;
    arAxisCtrl_gb[AxisNo.RackMotor].VelMode.Dec := CurrentData.Axes.RackMotor.Manual.JogDeceleration;
    arAxisCtrl_gb[AxisNo.RackMotor].VelMode.Jerk := CurrentData.Axes.RackMotor.Manual.JogJerk;
    arAxisCtrl_gb[AxisNo.RackMotor].VelMode.Velocity := CurrentData.Axes.RackMotor.Manual.JogVelocity;
    arAxisCtrl_gb[AxisNo.RackMotor].Admin._OpMode.en := E_AXIS_MODE.ModeVel;
ELSIF StorageManualCommand.RackMotor.Axis.JOG.MoveBWD AND AllowRackMotor THEN
    arAxisCtrl_gb[AxisNo.RackMotor].VelMode.Acc := CurrentData.Axes.RackMotor.Manual.JogAcceleration;
    arAxisCtrl_gb[AxisNo.RackMotor].VelMode.Dec := CurrentData.Axes.RackMotor.Manual.JogDeceleration;
    arAxisCtrl_gb[AxisNo.RackMotor].VelMode.Jerk := CurrentData.Axes.RackMotor.Manual.JogJerk;
    arAxisCtrl_gb[AxisNo.RackMotor].VelMode.Velocity := CurrentData.Axes.RackMotor.Manual.JogVelocity * -1;
    arAxisCtrl_gb[AxisNo.RackMotor].Admin._OpMode.en := E_AXIS_MODE.ModeVel;
ELSIF StorageManualCommand.RackMotor.Axis.PTP.Enable AND AllowRackMotor THEN
    arAxisCtrl_gb[AxisNo.RackMotor].PosMode.Acc := CurrentData.Axes.RackMotor.Manual.PtpAcceleration;
    arAxisCtrl_gb[AxisNo.RackMotor].PosMode.Dec := CurrentData.Axes.RackMotor.Manual.PtpDeceleration;
    arAxisCtrl_gb[AxisNo.RackMotor].PosMode.Jerk := CurrentData.Axes.RackMotor.Manual.PtpJerk;
    arAxisCtrl_gb[AxisNo.RackMotor].PosMode.Velocity := CurrentData.Axes.RackMotor.Manual.PtpVelocity;
    arAxisCtrl_gb[AxisNo.RackMotor].PosMode.Position := CurrentData.Axes.RackMotor.Manual.PtpPosition;
    arAxisCtrl_gb[AxisNo.RackMotor].Admin._OpMode.en := ModePosAbs;
ELSIF StorageManualCommand.RackMotor.Axis.Homing.Execute AND AllowRackMotor THEN
    arAxisCtrl_gb[AxisNo.RackMotor].SetupMode.eHomingMode := E_HomingMode._17_Neg_LimitOutterRight;
    arAxisCtrl_gb[AxisNo.RackMotor].SetupMode.FastVelo := CurrentData.Axes.RackMotor.Homing.FastVelo;
    arAxisCtrl_gb[AxisNo.RackMotor].SetupMode.SlowVelo := CurrentData.Axes.RackMotor.Homing.SlowVelo;
    arAxisCtrl_gb[AxisNo.RackMotor].SetupMode.lrOffset := CurrentData.Axes.RackMotor.Homing.Offset;
    arAxisCtrl_gb[AxisNo.RackMotor].SetupMode.lrSetPosition := CurrentData.Axes.RackMotor.Homing.SetAbsolutePosition;
    arAxisCtrl_gb[AxisNo.RackMotor].SetupMode.stPosBiasParameter.bSetPostionBias := TRUE;
    arAxisCtrl_gb[AxisNo.RackMotor].Admin._OpMode.en := ModeHoming;
ELSIF (TableMove.xBusy OR StorageService.AutoMode_AddBoxes.Status.Busy) AND AllowRackMotor THEN
    arAxisCtrl_gb[AxisNo.RackMotor].Admin._OpMode.en := ModePosAbs;
ELSIF fbStorageArea.fbBoxSupplyCtrl.Busy AND 
		fbStorageArea.fbBoxSupplyCtrl.AxisRackMotorBTNHomeRequest AND 
		AllowRackMotor THEN
	arAxisCtrl_gb[AxisNo.RackMotor].PosMode.Acc := CurrentData.Axes.RackMotor.HalfAuto.Acceleration;
	arAxisCtrl_gb[AxisNo.RackMotor].PosMode.Dec := CurrentData.Axes.RackMotor.HalfAuto.Deceleration;
	arAxisCtrl_gb[AxisNo.RackMotor].PosMode.Jerk := CurrentData.Axes.RackMotor.HalfAuto.Jerk;
	arAxisCtrl_gb[AxisNo.RackMotor].PosMode.Velocity := CurrentData.Axes.RackMotor.HalfAuto.Velocity;
	arAxisCtrl_gb[AxisNo.RackMotor].Admin._OpMode.en := ModePosAbs;
ELSE
    arAxisCtrl_gb[AxisNo.RackMotor].Admin.StopDeceleration := 1000;
    arAxisCtrl_gb[AxisNo.RackMotor].Admin._OpMode.en := E_AXIS_MODE.ModeAH;
END_IF

{endregion}
END_METHOD

METHOD M_Clearing
VAR
	CylinderIndex : INT;
	MotorIndex : INT;
	ServoIndex : INT;
END_VAR
VAR_INST
	AllCylinderNoError : BOOL := TRUE;
	AllMotorNoError : BOOL := TRUE;
	AllServoNoError : BOOL := TRUE;
END_VAR
// Disable all cylinder 
FOR CylinderIndex := 1 TO 53 DO
    Cylinder.arCylinder[CylinderIndex].xEnable := FALSE;
END_FOR

// Disable all motor
FOR MotorIndex := 1 TO 26 DO
    Motor.arMotor[MotorIndex].xEnable := FALSE;
END_FOR

// Check cylinder no error
FOR CylinderIndex := 1 TO 53 DO
    IF Cylinder.arCylinder[CylinderIndex].xError THEN
        AllCylinderNoError := FALSE;
        EXIT;
    END_IF
END_FOR

// Check motor no error
FOR MotorIndex := 1 TO 26 DO
    IF Motor.arMotor[MotorIndex].xError THEN
        AllMotorNoError := FALSE;
        EXIT;
    END_IF
END_FOR

FOR ServoIndex := 1 TO 7 DO
	IF arAxisCtrl_gb[ServoIndex].Admin.Axis.Status.Error THEN
		arAxisCtrl_gb[ServoIndex].Admin.ClearError := TRUE;
	END_IF
END_FOR
AllServoNoError := TRUE;
FOR ServoIndex := 1 TO 7 DO
    IF arAxisCtrl_gb[ServoIndex].Admin.Axis.Status.Error THEN
        AllServoNoError := FALSE;
        EXIT;
    END_IF
END_FOR
CASE eModeCurrent OF
    E_UnitMode.Manual:
        GVL_Machine.PackTags[UnitNo.Allocate].Command.UnitMode := E_UnitMode.Manual;
        GVL_Machine.PackTags[UnitNo.Allocate].Command.CntrlCmd := ePMLCommand_Clear;
        GVL_Machine.PackTags[UnitNo.Storage].Command.UnitMode := E_UnitMode.Manual;
        GVL_Machine.PackTags[UnitNo.Storage].Command.CntrlCmd := ePMLCommand_Clear;
        GVL_Machine.PackTags[UnitNo.Shipping].Command.UnitMode := E_UnitMode.Manual;
        GVL_Machine.PackTags[UnitNo.Shipping].Command.CntrlCmd := ePMLCommand_Clear;

        IF GVL_Machine.PackTags[UnitNo.Allocate].Status.StateCurrent = ePMLState_Stopped AND
            GVL_Machine.PackTags[UnitNo.Storage].Status.StateCurrent = ePMLState_Stopped AND
            GVL_Machine.PackTags[UnitNo.Shipping].Status.StateCurrent = ePMLState_Stopped THEN
            IF AllCylinderNoError AND AllMotorNoError AND AllServoNoError THEN
                M_StateComplete();
            END_IF
        END_IF

    E_UnitMode.Auto: ;
        GVL_Machine.PackTags[UnitNo.Allocate].Command.UnitMode := E_UnitMode.Auto;
        GVL_Machine.PackTags[UnitNo.Allocate].Command.CntrlCmd := ePMLCommand_Clear;
        GVL_Machine.PackTags[UnitNo.Storage].Command.UnitMode := E_UnitMode.Auto;
        GVL_Machine.PackTags[UnitNo.Storage].Command.CntrlCmd := ePMLCommand_Clear;
        GVL_Machine.PackTags[UnitNo.Shipping].Command.UnitMode := E_UnitMode.Auto;
        GVL_Machine.PackTags[UnitNo.Shipping].Command.CntrlCmd := ePMLCommand_Clear;

        IF GVL_Machine.PackTags[UnitNo.Allocate].Status.StateCurrent = ePMLState_Stopped AND
            GVL_Machine.PackTags[UnitNo.Storage].Status.StateCurrent = ePMLState_Stopped AND
            GVL_Machine.PackTags[UnitNo.Shipping].Status.StateCurrent = ePMLState_Stopped THEN
            IF AllCylinderNoError AND AllMotorNoError AND AllServoNoError THEN
                M_StateComplete();
            END_IF
        END_IF
END_CASE
END_METHOD

METHOD PRIVATE M_ClearOutput : BOOL
VAR_INPUT
END_VAR
VAR
	SpaceOutput : ST_OutputTable;
END_VAR
OUTPUT := SpaceOutput;
M_ClearOutput := true;
END_METHOD

METHOD M_Complete
M_StateComplete();
END_METHOD

METHOD M_Completing
M_StateComplete();
END_METHOD

METHOD M_Execute
//M_StateComplete();
CASE eModeCurrent OF
    E_UnitMode.Manual:
			M_Manual_Cylinder();
			M_Manual_Axes();
			M_Manual_Motor();
			M_HalfAuto_TableMove();
			IF NOT fbMachineHoming.xBusy THEN
				M_ManualAllocateHoming();
				M_ManualStorageHoming();
				M_ManualShippingHoming();
			END_IF
			M_ManualMachineHome();
			
    E_UnitMode.Auto:
			M_Auto_Axes();
  
END_CASE
//fbAllocateArea.A00_Service();
M_StroageRobotSafeCheck();
IF ErrorTableInitDone THEN
	M_General_AlarmRegister();
END_IF
END_METHOD

METHOD M_General_AlarmRegister : BOOL
VAR_INPUT
END_VAR
VAR
END_VAR
VAR_INST
	bTest 		  : ARRAY[1..200] OF BOOL;
	SafeDoorsOpen : ARRAY[0..20] OF BOOL;
END_VAR
/////  Category ==> 0 :machine Area ,1: StorageArea ,2: AllocateArea ,3: ShippingArea 

// E-Stop
RegisterAlarm(Trigger := Allocate_Estop, 								ID := 001,value := E_Severity.Level7, Message := 'Allocate Estop has trig', Category := 2);
RegisterAlarm(Trigger := Storage_EStop, 								ID := 002,value := E_Severity.Level7, Message := 'Storage Estop has trig', Category := 1);
RegisterAlarm(Trigger := FanucRobot.List.StorageRobot.E_Stop_Output,	ID := 003,value := E_Severity.Level7,Message := 'Storage robot Estop has trig',Category := 1);
RegisterAlarm(Trigger := FanucRobot.List.ShippingRobot.E_Stop_Output,	ID := 004,value := E_Severity.Level7,Message := 'Shipping robot Estop has trig',Category := 1);

//AirPressure
bStorage_AirPressure := NOT( BIT_TO_BOOL( INPUT.bStorage_AirPressure_Ready) ) OR  bTest2;
RegisterAlarm(Trigger := bStorage_AirPressure,							ID := 005,value := E_Severity.Level7,Message := 'Low AirPressure ',Category := 1);


//Homing Service
RegisterAlarm(Trigger := fbMachineHoming.xError,				ID := 11,value := E_Severity.Level4,Message := fbMachineHoming.ErrorMsg,Category := 0);
RegisterAlarm(Trigger := fbStorageArea.fbStorageHoming.xError,	ID := 12,value := E_Severity.Level4,Message := fbStorageArea.fbStorageHoming.ErrorMsg,Category := 1);
RegisterAlarm(Trigger := fballocateArea.fballocateHome.xError,	ID := 13,value := E_Severity.Level4,Message := fballocateArea.fballocateHome.ErrorMsg,Category := 2);
RegisterAlarm(Trigger := fbShippingArea.fbShippingHoming.xError,ID := 14,value := E_Severity.Level4,Message :=fbShippingArea.fbShippingHoming.ErrorMsg,Category := 3);
//Machine Area Service


//Storage Area Service
RegisterAlarm(Trigger := fbStorageArea.fbWarehouse.fbReloadBox.Error,				ID := 21,value := E_Severity.Level4,Message := fbStorageArea.fbWarehouse.fbReloadBox.Status,			Category := 1);
RegisterAlarm(Trigger := fbStorageArea.fbWarehouse.fbFeedInBox.Error,				ID := 22,value := E_Severity.Level4,Message := fbStorageArea.fbWarehouse.fbFeedInBox.Status,			Category := 1);
RegisterAlarm(Trigger := fbStorageArea.fbAddBoxes.Error ,							ID := 23,value := E_Severity.Level4,Message := fbStorageArea.fbAddBoxes.Status,							Category := 1);
RegisterAlarm(Trigger := fbStorageArea.fbBoxSupplyCtrl.Error ,						ID := 24,value := E_Severity.Level4,Message := fbStorageArea.fbBoxSupplyCtrl.Status,					Category := 1);
RegisterAlarm(Trigger := fbStorageArea.fbFeedInEmptyBoxWithRobot.Error ,			ID := 25,value := E_Severity.Level4,Message := fbStorageArea.fbFeedInEmptyBoxWithRobot.Status,			Category := 1);
RegisterAlarm(Trigger := fbStorageArea.fbReloadRoundBeltBoxWithRobot.Error ,		ID := 26,value := E_Severity.Level4,Message := fbStorageArea.fbReloadRoundBeltBoxWithRobot.Status,		Category := 1);
RegisterAlarm(Trigger := fbStorageArea.fbRobotAbsMove.Error ,						ID := 27,value := E_Severity.Level4,Message := fbStorageArea.fbRobotAbsMove.Status,						Category := 1);
RegisterAlarm(Trigger := fbStorageArea.fbRobotRegionMove_AllocatedConveyor.Error ,	ID := 28,value := E_Severity.Level4,Message := fbStorageArea.fbRobotRegionMove_AllocatedConveyor.Status,Category := 1);
RegisterAlarm(Trigger := fbStorageArea.fbRobotRegionMove_BufferArea.Error ,			ID := 29,value := E_Severity.Level4,Message := fbStorageArea.fbRobotRegionMove_BufferArea.Status,		Category := 1);
RegisterAlarm(Trigger := fbStorageArea.fbRobotRegionMove_FeedInConveyor.Error ,		ID := 30,value := E_Severity.Level4,Message := fbStorageArea.fbRobotRegionMove_FeedInConveyor.Status,	Category := 1);
RegisterAlarm(Trigger := fbStorageArea.fbRobotRegionMove_PullOutConveyor.Error ,	ID := 31,value := E_Severity.Level4,Message := fbStorageArea.fbRobotRegionMove_PullOutConveyor.Status,	Category := 1);
RegisterAlarm(Trigger := fbStorageArea.fbRobotRegionMove_RoundBelt.Error ,			ID := 32,value := E_Severity.Level4,Message := fbStorageArea.fbRobotRegionMove_RoundBelt.Status,		Category := 1);
RegisterAlarm(Trigger := fbStorageArea.fbUpperFeedInConveyor.Error ,				ID := 33,value := E_Severity.Level4,Message := fbStorageArea.fbUpperFeedInConveyor.Status,				Category := 1);
RegisterAlarm(Trigger := fbStorageArea.fbWareHouseWithRobotMove.Error ,				ID := 34,value := E_Severity.Level4,Message := fbStorageArea.fbWareHouseWithRobotMove.Status,			Category := 1);

//Storage Cabinet Internal Service
RegisterAlarm(Trigger := fbStorageArea.fbWarehouse.fbFeedInBox.Error, 				ID := 50,value := E_Severity.Level3,Message := fbStorageArea.fbWarehouse.fbFeedInBox.Status,			Category := 1);
RegisterAlarm(Trigger := fbStorageArea.fbWarehouse.fbReloadBox.Error, 				ID := 51,value := E_Severity.Level3,Message := fbStorageArea.fbWarehouse.fbReloadBox.Status,			Category := 1);

//Allocate Area Service
RegisterAlarm(Trigger := fbAllocateArea.fb_AllocateBatchMode.Error ,				ID := 35,value := E_Severity.Level3,Message := fbAllocateArea.fb_AllocateBatchMode.Status,			Category := 2);
RegisterAlarm(Trigger := fbAllocateArea.fb_AllocateBatchMode_Reverse.Error ,		ID := 36,value := E_Severity.Level3,Message := fbAllocateArea.fb_AllocateBatchMode_Reverse.Status,	Category := 2);
RegisterAlarm(Trigger := fbAllocateArea.fbDifferentCVCamera.xError ,				ID := 37,value := E_Severity.Level3,Message := fbAllocateArea.fbDifferentCVCamera.ErrorMsg,			Category := 2);
RegisterAlarm(Trigger := fbAllocateArea.fbOutRobot_BoxMoveReverse.Error ,			ID := 38,value := E_Severity.Level3,Message := fbAllocateArea.fbOutRobot_BoxMoveReverse.Status,		Category := 2);
RegisterAlarm(Trigger := fbAllocateArea.fbOutRobot_EmptyBoxMove.Error ,				ID := 39,value := E_Severity.Level3,Message := fbAllocateArea.fbOutRobot_EmptyBoxMove.Status,		Category := 2);
RegisterAlarm(Trigger := fbAllocateArea.fbOutRobot_RareBoxMove.Error ,				ID := 40,value := E_Severity.Level3,Message := fbAllocateArea.fbOutRobot_RareBoxMove.Status,		Category := 2);
RegisterAlarm(Trigger := fbAllocateArea.fbPulloutCV.Error ,							ID := 41,value := E_Severity.Level3,Message := fbAllocateArea.fbPulloutCV.Status,					Category := 2);
RegisterAlarm(Trigger := fbAllocateArea.RoundBeltControl.xError ,					ID := 42,value := E_Severity.Level3,Message := fbAllocateArea.RoundBeltControl.ErrorMsg,			Category := 2);
RegisterAlarm(Trigger := fbAllocateArea.fbSameSizeCVCamera.xError ,					ID := 43,value := E_Severity.Level3,Message := fbAllocateArea.fbSameSizeCVCamera.ErrorMsg,			Category := 2);
RegisterAlarm(Trigger := fbAllocateArea.TurnTableControl.xError ,					ID := 44,value := E_Severity.Level3,Message := fbAllocateArea.TurnTableControl.ErrorMsg,			Category := 2);
RegisterAlarm(Trigger := fbAllocateArea.fbOutRobot_TurnTableToRoundBelt.Error ,		ID := 45,value := E_Severity.Level3,Message := fbAllocateArea.fbOutRobot_TurnTableToRoundBelt.Status,Category := 2);
RegisterAlarm(Trigger := fbAllocateArea.fbAllocateRobotNeedlingMove.xError, id:= 49,value:= E_Severity.Level3,Message:=fbAllocateArea.fbAllocateRobotNeedlingMove.ErrorMsg,				Category :=2);

//Shipping Area Service
RegisterAlarm(Trigger := fbShippingArea.fbShippingRobot_Left.Error ,			ID := 46,value := E_Severity.Level3,Message := fbShippingArea.fbShippingRobot_Left.Status,Category := 3);
RegisterAlarm(Trigger := fbShippingArea.fbShippingRobot_Right.Error ,			ID := 47,value := E_Severity.Level3,Message := fbShippingArea.fbShippingRobot_Right.Status,Category := 3);
RegisterAlarm(Trigger := fbShippingArea.fbShippingRobot_TransmitCVEnd.Error ,	ID := 48,value := E_Severity.Level3,Message := fbShippingArea.fbShippingRobot_TransmitCVEnd.Status,Category := 3);



// Cylinder Allocate Area component
RegisterAlarm(Trigger := Cylinder.List.fbAllocateRobot_LeftClamp1.xError,		ID := 101,value := E_Severity.Level2,Message := Cylinder.List.fbAllocateRobot_LeftClamp1.ErrorMsg,Category := 2);
RegisterAlarm(Trigger := Cylinder.List.fbAllocateRobot_LeftClamp2.xError,		ID := 102,value := E_Severity.Level2,Message := Cylinder.List.fbAllocateRobot_LeftClamp2.ErrorMsg,Category := 2);
RegisterAlarm(Trigger := Cylinder.List.fbAllocateRobot_LeftVert1.xError,		ID := 103,value := E_Severity.Level2,Message := Cylinder.List.fbAllocateRobot_LeftVert1.ErrorMsg,Category := 2);
RegisterAlarm(Trigger := Cylinder.List.fbAllocateRobot_LeftVert2.xError,		ID := 104,value := E_Severity.Level2,Message := Cylinder.List.fbAllocateRobot_LeftVert2.ErrorMsg,Category := 2);
RegisterAlarm(Trigger := Cylinder.List.fbAllocateRobot_RightClamp1.xError,		ID := 105,value := E_Severity.Level2,Message := Cylinder.List.fbAllocateRobot_RightClamp1.ErrorMsg,Category := 2);
RegisterAlarm(Trigger := Cylinder.List.fbAllocateRobot_RightClamp2.xError,		ID := 106,value := E_Severity.Level2,Message := Cylinder.List.fbAllocateRobot_RightClamp2.ErrorMsg,Category := 2);
RegisterAlarm(Trigger := Cylinder.List.fbAllocateRobot_RightVert1.xError,		ID := 107,value := E_Severity.Level2,Message := Cylinder.List.fbAllocateRobot_RightVert1.ErrorMsg,Category := 2);
RegisterAlarm(Trigger := Cylinder.List.fbAllocateRobot_RightVert2.xError,		ID := 108,value := E_Severity.Level2,Message := Cylinder.List.fbAllocateRobot_RightVert2.ErrorMsg,Category := 2);
RegisterAlarm(Trigger := Cylinder.List.fbDifferentSizeCV_Block1.xError,			ID := 109,value := E_Severity.Level2,Message := Cylinder.List.fbDifferentSizeCV_Block1.ErrorMsg,Category := 2);
RegisterAlarm(Trigger := Cylinder.List.fbRoundBelt_WorkZone_Press.xError,		ID := 110,value := E_Severity.Level2,Message := Cylinder.List.fbRoundBelt_WorkZone_Press.ErrorMsg,Category := 2);
RegisterAlarm(Trigger := Cylinder.List.fbRoundBelt_WorkZone_Plug.xError,		ID := 111,value := E_Severity.Level2,Message := Cylinder.List.fbRoundBelt_WorkZone_Plug.ErrorMsg,Category := 2);
RegisterAlarm(Trigger := Cylinder.List.fbRoundBelt_ChargeZone_Plug.xError,		ID := 112,value := E_Severity.Level2,Message := Cylinder.List.fbRoundBelt_ChargeZone_Plug.ErrorMsg,Category := 2);
RegisterAlarm(Trigger := Cylinder.List.fbRoundBelt_TransmitCVZone_Plug.xError,	ID := 113,value := E_Severity.Level2,Message := Cylinder.List.fbRoundBelt_TransmitCVZone_Plug.ErrorMsg,Category := 2);
RegisterAlarm(Trigger := Cylinder.List.fbOutRobot_AsideVert.xError,				ID := 114,value := E_Severity.Level2,Message := Cylinder.List.fbOutRobot_AsideVert.ErrorMsg,Category := 2);
RegisterAlarm(Trigger := Cylinder.List.fbOutRobot_BsideVert.xError,				ID := 115,value := E_Severity.Level2,Message := Cylinder.List.fbOutRobot_BsideVert.ErrorMsg,Category := 2);
RegisterAlarm(Trigger := Cylinder.List.fbOutRobot_AsideClamp.xError,			ID := 116,value := E_Severity.Level2,Message := Cylinder.List.fbOutRobot_AsideClamp.ErrorMsg,Category := 2);
RegisterAlarm(Trigger := Cylinder.List.fbOutRobot_BsideClamp.xError,			ID := 117,value := E_Severity.Level2,Message := Cylinder.List.fbOutRobot_BsideClamp.ErrorMsg,Category := 2);
RegisterAlarm(Trigger := Cylinder.List.fbTransmitCV_CamaraHoriz.xError,			ID := 118,value := E_Severity.Level2,Message := Cylinder.List.fbTransmitCV_CamaraHoriz.ErrorMsg,Category := 2);
RegisterAlarm(Trigger := Cylinder.List.fbDifferentSizeCV_Press2.xError,			ID := 119,value := E_Severity.Level2,Message := Cylinder.List.fbDifferentSizeCV_Press2.ErrorMsg,Category := 2);
RegisterAlarm(Trigger := Cylinder.List.fbDifferentSizeCV_Press1.xError,			ID := 120,value := E_Severity.Level2,Message := Cylinder.List.fbDifferentSizeCV_Press1.ErrorMsg,Category := 2);
RegisterAlarm(Trigger := Cylinder.List.fbDifferentSizeCV_Block1.xError,			ID := 121,value := E_Severity.Level2,Message := Cylinder.List.fbDifferentSizeCV_Block1.ErrorMsg,Category := 2);
RegisterAlarm(Trigger := Cylinder.List.fbSameSizeCV_Press4.xError,				ID := 122,value := E_Severity.Level2,Message := Cylinder.List.fbSameSizeCV_Press4.ErrorMsg,Category := 2);
RegisterAlarm(Trigger := Cylinder.List.fbSameSizeCV_Press3.xError,				ID := 123,value := E_Severity.Level2,Message := Cylinder.List.fbSameSizeCV_Press3.ErrorMsg,Category := 2);
RegisterAlarm(Trigger := Cylinder.List.fbSameSizeCV_Press2.xError,				ID := 124,value := E_Severity.Level2,Message := Cylinder.List.fbSameSizeCV_Press2.ErrorMsg,Category := 2);
RegisterAlarm(Trigger := Cylinder.List.fbSameSizeCV_Press1.xError,				ID := 125,value := E_Severity.Level2,Message := Cylinder.List.fbSameSizeCV_Press1.ErrorMsg,Category := 2);
RegisterAlarm(Trigger := Cylinder.List.fbSameSizeCV_Block2.xError,				ID := 126,value := E_Severity.Level2,Message := Cylinder.List.fbSameSizeCV_Block2.ErrorMsg,Category := 2);
RegisterAlarm(Trigger := Cylinder.List.fbSameSizeCV_Block1.xError,				ID := 127,value := E_Severity.Level2,Message := Cylinder.List.fbSameSizeCV_Block1.ErrorMsg,Category := 2);
RegisterAlarm(Trigger := Cylinder.List.fbPullOutCV_AsidePress1.xError,			ID := 128,value := E_Severity.Level2,Message := Cylinder.List.fbPullOutCV_AsidePress1.ErrorMsg,Category := 2);
RegisterAlarm(Trigger := Cylinder.List.fbPullOutCV_AsidePress2.xError,			ID := 129,value := E_Severity.Level2,Message := Cylinder.List.fbPullOutCV_AsidePress2.ErrorMsg,Category := 2);
RegisterAlarm(Trigger := Cylinder.List.fbPullOutCV_AsideBlock.xError,			ID := 130,value := E_Severity.Level2,Message := Cylinder.List.fbPullOutCV_AsideBlock.ErrorMsg,Category := 2);
RegisterAlarm(Trigger := Cylinder.List.fbPullOutCV_BsidePress1.xError,			ID := 131,value := E_Severity.Level2,Message := Cylinder.List.fbPullOutCV_BsidePress1.ErrorMsg,Category := 2);
RegisterAlarm(Trigger := Cylinder.List.fbPullOutCV_BsidePress2.xError,			ID := 132,value := E_Severity.Level2,Message := Cylinder.List.fbPullOutCV_BsidePress2.ErrorMsg,Category := 2);
RegisterAlarm(Trigger := Cylinder.List.fbPullOutCV_BsideBlock.xError,			ID := 133,value := E_Severity.Level2,Message := Cylinder.List.fbPullOutCV_BsideBlock.ErrorMsg,Category := 2);

// Cyliner Storage Area component
RegisterAlarm(Trigger := Cylinder.List.fbUpCV_FeedInPress1.xError,				ID := 134,value := E_Severity.Level2,Message := Cylinder.List.fbUpCV_FeedInPress1.ErrorMsg,Category := 1);
RegisterAlarm(Trigger := Cylinder.List.fbUpCV_FeedInPress2.xError,				ID := 135,value := E_Severity.Level2,Message := Cylinder.List.fbUpCV_FeedInPress2.ErrorMsg,Category := 1);
RegisterAlarm(Trigger := Cylinder.List.fbUpCV_DiameterPress.xError,				ID := 136,value := E_Severity.Level2,Message := Cylinder.List.fbUpCV_DiameterPress.ErrorMsg,Category := 1);
RegisterAlarm(Trigger := Cylinder.List.fbUpCV_CamaraPress1.xError,				ID := 137,value := E_Severity.Level2,Message := Cylinder.List.fbUpCV_CamaraPress1.ErrorMsg,Category := 1);
RegisterAlarm(Trigger := Cylinder.List.fbUpCV_CamaraPress2.xError,				ID := 138,value := E_Severity.Level2,Message := Cylinder.List.fbUpCV_CamaraPress2.ErrorMsg,Category := 1);
RegisterAlarm(Trigger := Cylinder.List.fbUpCV_CamaraPress3.xError,				ID := 139,value := E_Severity.Level2,Message := Cylinder.List.fbUpCV_CamaraPress3.ErrorMsg,Category := 1);
RegisterAlarm(Trigger := Cylinder.List.fbUpCV_CamaraPress4.xError,				ID := 140,value := E_Severity.Level2,Message := Cylinder.List.fbUpCV_CamaraPress4.ErrorMsg,Category := 1);
RegisterAlarm(Trigger := Cylinder.List.fbUpCV_Block1.xError,					ID := 141,value := E_Severity.Level2,Message := Cylinder.List.fbUpCV_Block1.ErrorMsg,Category := 1);
RegisterAlarm(Trigger := Cylinder.List.fbUpCV_Block2.xError,					ID := 142,value := E_Severity.Level2,Message := Cylinder.List.fbUpCV_Block2.ErrorMsg,Category := 1);
RegisterAlarm(Trigger := Cylinder.List.fbUpCV_Block3.xError,					ID := 143,value := E_Severity.Level2,Message := Cylinder.List.fbUpCV_Block3.ErrorMsg,Category := 1);
RegisterAlarm(Trigger := Cylinder.List.fbUpCV_DiameterHoriz.xError,				ID := 144,value := E_Severity.Level2,Message := Cylinder.List.fbUpCV_DiameterHoriz.ErrorMsg,Category := 1);
RegisterAlarm(Trigger := Cylinder.List.fbUpCV_DiameterVert.xError,				ID := 145,value := E_Severity.Level2,Message := Cylinder.List.fbUpCV_DiameterVert.ErrorMsg,Category := 1);
RegisterAlarm(Trigger := Cylinder.List.fbUpCV_DiameterClamp.xError,				ID := 146,value := E_Severity.Level2,Message := Cylinder.List.fbUpCV_DiameterClamp.ErrorMsg,Category := 1);
RegisterAlarm(Trigger := Cylinder.List.fbStackPush.xError,						ID := 147,value := E_Severity.Level2,Message := Cylinder.List.fbStackPush.ErrorMsg,Category := 1);
RegisterAlarm(Trigger := Cylinder.List.fbLowCV_Press1.xError,					ID := 148,value := E_Severity.Level2,Message := Cylinder.List.fbLowCV_Press1.ErrorMsg,Category := 1);
RegisterAlarm(Trigger := Cylinder.List.fbLowCV_Press2.xError,					ID := 149,value := E_Severity.Level2,Message := Cylinder.List.fbLowCV_Press2.ErrorMsg,Category := 1);
RegisterAlarm(Trigger := Cylinder.List.fbLowCV_Press3.xError,					ID := 150,value := E_Severity.Level2,Message := Cylinder.List.fbLowCV_Press3.ErrorMsg,Category := 1);
RegisterAlarm(Trigger := Cylinder.List.fbLowCV_Press4.xError,					ID := 151,value := E_Severity.Level2,Message := Cylinder.List.fbLowCV_Press4.ErrorMsg,Category := 1);
RegisterAlarm(Trigger := Cylinder.List.fbLowCV_Block1.xError,					ID := 152,value := E_Severity.Level2,Message := Cylinder.List.fbLowCV_Block1.ErrorMsg,Category := 1);
RegisterAlarm(Trigger := Cylinder.List.fbLowCV_Block2.xError,					ID := 153,value := E_Severity.Level2,Message := Cylinder.List.fbLowCV_Block2.ErrorMsg,Category := 1);

// Robot Error
//RegisterAlarm(Trigger := fanucrobot.List.StorageRobot.Error,					ID := 158,value := E_Severity.Level5,Message := fanucrobot.List.StorageRobot.ErrMsg,Category:=1);
//RegisterAlarm(Trigger := fanucrobot.List.ShippingRobot.Error,					ID := 159,value := E_Severity.Level5,Message := fanucrobot.List.ShippingRobot.ErrMsg,Category:=1);


// Servo Error
RegisterAlarm(Trigger := arAxisCtrl_gb[AxisNo.TurnTable].Admin.Axis.Status.Error,ID := 201,value := E_Severity.Level6,Message := 'TurnTable axis has Error',Category := 2);
RegisterAlarm(Trigger := arAxisCtrl_gb[AxisNo.RoundBelt].Admin.Axis.Status.Error,ID := 202,value := E_Severity.Level6,Message := 'Roundbelt axis has Error',Category := 2);
RegisterAlarm(Trigger := arAxisCtrl_gb[AxisNo.Allocate_X].Admin.Axis.Status.Error,ID := 203,value := E_Severity.Level6,Message := 'Allocate_X axis has Error',Category := 2);
RegisterAlarm(Trigger := arAxisCtrl_gb[AxisNo.Allocate_Y].Admin.Axis.Status.Error,ID := 204,value := E_Severity.Level6,Message := 'Allocate_Y axis has Error',Category := 2);
RegisterAlarm(Trigger := arAxisCtrl_gb[AxisNo.OutRobot_X].Admin.Axis.Status.Error,ID := 205,value := E_Severity.Level6,Message := 'OutRobot_X axis has Error',Category := 2);
RegisterAlarm(Trigger := arAxisCtrl_gb[AxisNo.OutRobot_Y].Admin.Axis.Status.Error,ID := 206,value := E_Severity.Level6,Message := 'OutRobot_Y axis has Error',Category := 2);
RegisterAlarm(Trigger := arAxisCtrl_gb[AxisNo.RackMotor].Admin.Axis.Status.Error,ID := 207,value := E_Severity.Level6,Message := 'RackMotor axis has Error',Category := 1);

// ModbusRTU 
RegisterAlarm(Trigger := ComModbusRTU.fb_Warehouse_Modbus[0].Error,ID := 300,value := E_Severity.Level2,Message := ComModbusRTU.fb_Warehouse_Modbus[0].Status,Category := 1);
RegisterAlarm(Trigger := ComModbusRTU.fb_Warehouse_Modbus[1].Error,ID := 301,value := E_Severity.Level2,Message := ComModbusRTU.fb_Warehouse_Modbus[1].Status,Category := 1);
RegisterAlarm(Trigger := ComModbusRTU.fb_Warehouse_Modbus[2].Error,ID := 302,value := E_Severity.Level2,Message := ComModbusRTU.fb_Warehouse_Modbus[2].Status,Category := 1);
RegisterAlarm(Trigger := ComModbusRTU.fb_Warehouse_Modbus[3].Error,ID := 303,value := E_Severity.Level2,Message := ComModbusRTU.fb_Warehouse_Modbus[3].Status,Category := 1);


//Safe Door
SafeDoorsOpen[1] 	:=  NOT INPUT.bSafetyDoor1   AND NOT GVL_HMI.Setup.Mechanical.stSafetyByPass.SafeDoorByPass;	 
SafeDoorsOpen[2] 	:=  NOT INPUT.bSafetyDoor2   AND NOT GVL_HMI.Setup.Mechanical.stSafetyByPass.SafeDoorByPass;	 
SafeDoorsOpen[3] 	:=  NOT INPUT.bSafetyDoor3   AND NOT GVL_HMI.Setup.Mechanical.stSafetyByPass.SafeDoorByPass;	 
SafeDoorsOpen[4] 	:=  NOT INPUT.bSafetyDoor4   AND NOT GVL_HMI.Setup.Mechanical.stSafetyByPass.SafeDoorByPass;
SafeDoorsOpen[5] 	:=  NOT INPUT.bSafetyDoor5   AND NOT GVL_HMI.Setup.Mechanical.stSafetyByPass.SafeDoorByPass;	 
SafeDoorsOpen[6] 	:=  NOT INPUT.bSafetyDoor6   AND NOT GVL_HMI.Setup.Mechanical.stSafetyByPass.SafeDoorByPass;	 
SafeDoorsOpen[7] 	:=  NOT INPUT.bSafetyDoor7   AND NOT GVL_HMI.Setup.Mechanical.stSafetyByPass.SafeDoorByPass;	 
SafeDoorsOpen[8] 	:=  NOT INPUT.bSafetyDoor8   AND NOT GVL_HMI.Setup.Mechanical.stSafetyByPass.SafeDoorByPass;	 
SafeDoorsOpen[9] 	:=  NOT INPUT.bSafetyDoor9   AND NOT GVL_HMI.Setup.Mechanical.stSafetyByPass.SafeDoorByPass;	 
SafeDoorsOpen[10] 	:=  NOT INPUT.bSafetyDoor10   AND NOT GVL_HMI.Setup.Mechanical.stSafetyByPass.SafeDoorByPass;	 
SafeDoorsOpen[11] 	:=  NOT INPUT.bSafetyDoor11   AND NOT GVL_HMI.Setup.Mechanical.stSafetyByPass.SafeDoorByPass;	 
SafeDoorsOpen[12] 	:=  NOT INPUT.bSafetyDoor12   AND NOT GVL_HMI.Setup.Mechanical.stSafetyByPass.SafeDoorByPass;	 
SafeDoorsOpen[13] 	:=  NOT INPUT.bSafetyDoor13   AND NOT GVL_HMI.Setup.Mechanical.stSafetyByPass.SafeDoorByPass;	 
SafeDoorsOpen[14] 	:=  NOT INPUT.bSafetyDoor14   AND NOT GVL_HMI.Setup.Mechanical.stSafetyByPass.SafeDoorByPass;	 
SafeDoorsOpen[15] 	:=  NOT INPUT.bAllocate_Electrical_Cabinet_SafetyDoor   AND NOT GVL_HMI.Setup.Mechanical.stSafetyByPass.SafeDoorByPass;	 
SafeDoorsOpen[16] 	:=  NOT INPUT.bShippingRobot_ElectricalCabinet_SafetyDoor   AND NOT GVL_HMI.Setup.Mechanical.stSafetyByPass.SafeDoorByPass;	 
IF NOT GVL_HMI.Setup.Mechanical.stSafetyByPass.SafeDoorByPass THEN
	RegisterAlarm(Trigger := SafeDoorsOpen[1],  ID := 401, value := E_Severity.Level2, Message := 'Safe door1  Opened',  Category := 1); 
	RegisterAlarm(Trigger := SafeDoorsOpen[2],  ID := 402, value := E_Severity.Level2, Message := 'Safe door2  Opened',  Category := 1); 
	RegisterAlarm(Trigger := SafeDoorsOpen[3],  ID := 403, value := E_Severity.Level2, Message := 'Safe door3  Opened',  Category := 1); 
	RegisterAlarm(Trigger := SafeDoorsOpen[4],  ID := 404, value := E_Severity.Level2, Message := 'Safe door4  Opened',  Category := 1); 
	RegisterAlarm(Trigger := SafeDoorsOpen[5],  ID := 405, value := E_Severity.Level2, Message := 'Safe door5  Opened',  Category := 1); 
	RegisterAlarm(Trigger := SafeDoorsOpen[6],  ID := 406, value := E_Severity.Level2, Message := 'Safe door6  Opened',  Category := 1); 
	RegisterAlarm(Trigger := SafeDoorsOpen[7],  ID := 407, value := E_Severity.Level2, Message := 'Safe door7  Opened',  Category := 1); 
	RegisterAlarm(Trigger := SafeDoorsOpen[8],  ID := 408, value := E_Severity.Level2, Message := 'Safe door8  Opened',  Category := 1); 
	RegisterAlarm(Trigger := SafeDoorsOpen[9],	ID := 409, value := E_Severity.Level2, Message := 'Safe door9  Opened',  Category := 1); 
	RegisterAlarm(Trigger := SafeDoorsOpen[10],	ID := 410, value := E_Severity.Level2, Message := 'Safe door10  Opened',  Category := 1); 
	RegisterAlarm(Trigger := SafeDoorsOpen[11],	ID := 411, value := E_Severity.Level2, Message := 'Safe door11  Opened',  Category := 1); 
	RegisterAlarm(Trigger := SafeDoorsOpen[12],	ID := 412, value := E_Severity.Level2, Message := 'Safe doo12  Opened',  Category := 1); 
	RegisterAlarm(Trigger := SafeDoorsOpen[13],	ID := 413, value := E_Severity.Level2, Message := 'Safe doo13  Opened',  Category := 1); 
	RegisterAlarm(Trigger := SafeDoorsOpen[14],	ID := 414, value := E_Severity.Level2, Message := 'Safe door14  Opened',  Category := 1); 
	RegisterAlarm(Trigger := SafeDoorsOpen[15],	ID := 415, value := E_Severity.Level2, Message := 'Allocate_Electrical_Cabinet_SafetyDoor  Opened',  Category := 1); 
	RegisterAlarm(Trigger := SafeDoorsOpen[16],	ID := 416, value := E_Severity.Level2, Message := 'bShippingRobot_ElectricalCabinet_SafetyDoor  Opened',  Category := 1); 
END_IF

M_General_AlarmRegister := TRUE;
END_METHOD

METHOD M_GetCylinderError : BOOL
VAR_INPUT
END_VAR
VAR
	udiCylinderIndex : UDINT;
END_VAR
FOR udiCylinderIndex := 1 TO udiMax_CylinderNum DO
	IF Cylinder.arCylinder[udiCylinderIndex].xError THEN
		M_GetCylinderError := TRUE;
	END_IF
END_FOR
END_METHOD

METHOD M_HalfAuto_TableMove
VAR_INPUT
END_VAR
// TableMove service 
TableMove(
	xDone=> AllocateHalfAutoCommand.TableMove.Status.Done, 
	xBusy=> AllocateHalfAutoCommand.TableMove.Status.Busy, 
	xError=> AllocateHalfAutoCommand.TableMove.Status.Error, 
	xExecute:= AllocateHalfAutoCommand.TableMove.Ctrl.Execute, 
	xAbort:= AllocateHalfAutoCommand.TableMove.Ctrl.Abort,
	xReset :=  AllocateHalfAutoCommand.TableMove.Ctrl.Reset,
	Index:= AllocateHalfAutoCommand.TableMove.Ctrl.Index, 
	CurrentData:= CurrentData, 
	xAborted=> AllocateHalfAutoCommand.TableMove.Status.Aborted);
END_METHOD

METHOD M_Held
M_StateComplete();
END_METHOD

METHOD M_Holding
M_StateComplete();
END_METHOD

METHOD M_Idle
IF eModeCurrent = E_UnitMode.Auto THEN
	GVL_Machine.PackTags[UnitNo.Storage].Command.UnitMode := E_UnitMode.Auto;
	GVL_Machine.PackTags[UnitNo.Allocate].Command.UnitMode := E_UnitMode.Auto;
	GVL_Machine.PackTags[UnitNo.Shipping].Command.UnitMode := E_UnitMode.Auto;
ELSIF eModeCurrent = E_UnitMode.Manual THEN
	GVL_Machine.PackTags[UnitNo.Storage].Command.UnitMode := E_UnitMode.Manual;
	GVL_Machine.PackTags[UnitNo.Allocate].Command.UnitMode := E_UnitMode.Manual;
	GVL_Machine.PackTags[UnitNo.Shipping].Command.UnitMode := E_UnitMode.Manual;
END_IF

M_StateComplete();
END_METHOD

METHOD M_MachineHoming : BOOL
VAR_INPUT
END_VAR
fbMachineHoming.xExecute :=   Service_Handshake.MachineHome.HandShake.Execute;
fbMachineHoming.xAbort := Machine_Stop;

Service_Handshake.MachineHome.HandShake.Done := fbMachineHoming.xDone;
Service_Handshake.MachineHome.HandShake.Busy := fbMachineHoming.xBusy;
Service_Handshake.MachineHome.HandShake.Error := fbMachineHoming.xError;
END_METHOD

METHOD PRIVATE M_Manual_Axes
VAR_INPUT
END_VAR

VAR_INST
	AllowAllocateRobotMove : BOOL;
	AllowOutRobotMove : BOOL;
	AllowRoundBeltMove : BOOL;
	AllowTurnTable		:BOOL;
	AllowRackMotor		:BOOL;
END_VAR
// Safe check
AllowAllocateRobotMove := Cylinder.List.fbAllocateRobot_LeftVert1.InRearPosition AND
    Cylinder.List.fbAllocateRobot_LeftVert2.InRearPosition AND
    Cylinder.List.fbAllocateRobot_RightVert1.InRearPosition AND
    Cylinder.List.fbAllocateRobot_RightVert2.InRearPosition;

AllowOutRobotMove := Cylinder.List.fbOutRobot_AsideVert.InRearPosition AND Cylinder.List.fbOutRobot_BsideVert.InRearPosition;
AllowRoundBeltMove := Cylinder.List.fbRoundBelt_ChargeZone_Plug.InRearPosition AND
    Cylinder.List.fbRoundBelt_TransmitCVZone_Plug.InRearPosition AND
    Cylinder.List.fbRoundBelt_WorkZone_Plug.InRearPosition AND
    Cylinder.List.fbRoundBelt_WorkZone_Press.InRearPosition AND
    AllowAllocateRobotMove AND
    AllowOutRobotMove 
	AND NOT FanucRobot.List.StorageRobot.BZoneInWork AND NOT FanucRobot.List.StorageRobot.Bzone_AllowWork;

AllowTurnTable := Cylinder.List.fbTurntable_Press.InRearPosition;
AllowRackMotor := Cylinder.List.fbStackPush.InRearPosition;

// Axis controll
{region "AllocateRobot AxisX"}

IF AllocateManualCommand.AllocatedRobot.AxisX.JOG.MoveFWD AND AllowAllocateRobotMove  THEN
    arAxisCtrl_gb[AxisNo.Allocate_X].VelMode.Acc := CurrentData.Axes.Allocate_X.Manual.JogAcceleration;
    arAxisCtrl_gb[AxisNo.Allocate_X].VelMode.Dec := CurrentData.Axes.Allocate_X.Manual.JogDeceleration;
    arAxisCtrl_gb[AxisNo.Allocate_X].VelMode.Jerk := CurrentData.Axes.Allocate_X.Manual.JogJerk;
    arAxisCtrl_gb[AxisNo.Allocate_X].VelMode.Velocity := CurrentData.Axes.Allocate_X.Manual.JogVelocity;
    arAxisCtrl_gb[AxisNo.Allocate_X].Admin._OpMode.en := E_AXIS_MODE.ModeVel;
ELSIF AllocateManualCommand.AllocatedRobot.AxisX.JOG.MoveBWD AND AllowAllocateRobotMove THEN
    arAxisCtrl_gb[AxisNo.Allocate_X].VelMode.Acc := CurrentData.Axes.Allocate_X.Manual.JogAcceleration;
    arAxisCtrl_gb[AxisNo.Allocate_X].VelMode.Dec := CurrentData.Axes.Allocate_X.Manual.JogDeceleration;
    arAxisCtrl_gb[AxisNo.Allocate_X].VelMode.Jerk := CurrentData.Axes.Allocate_X.Manual.JogJerk;
    arAxisCtrl_gb[AxisNo.Allocate_X].VelMode.Velocity := CurrentData.Axes.Allocate_X.Manual.JogVelocity * -1;
    arAxisCtrl_gb[AxisNo.Allocate_X].Admin._OpMode.en := E_AXIS_MODE.ModeVel;
ELSIF AllocateManualCommand.AllocatedRobot.AxisX.PTP.Enable  AND AllowAllocateRobotMove THEN
    arAxisCtrl_gb[AxisNo.Allocate_X].PosMode.Acc := CurrentData.Axes.Allocate_X.Manual.PtpAcceleration;
    arAxisCtrl_gb[AxisNo.Allocate_X].PosMode.Dec := CurrentData.Axes.Allocate_X.Manual.PtpDeceleration;
    arAxisCtrl_gb[AxisNo.Allocate_X].PosMode.Jerk := CurrentData.Axes.Allocate_X.Manual.PtpJerk;
    arAxisCtrl_gb[AxisNo.Allocate_X].PosMode.Velocity := CurrentData.Axes.Allocate_X.Manual.PtpVelocity;
    arAxisCtrl_gb[AxisNo.Allocate_X].PosMode.Position := CurrentData.Axes.Allocate_X.Manual.PtpPosition;
    arAxisCtrl_gb[AxisNo.Allocate_X].Admin._OpMode.en := ModePosAbs;
ELSIF (AllocateManualCommand.AllocatedRobot.AxisX.Homing.Execute OR  fbAllocateArea.fbAllocateHome.AxisHomingRequest)  AND AllowAllocateRobotMove THEN
    arAxisCtrl_gb[AxisNo.Allocate_X].SetupMode.eHomingMode := E_HomingMode._17_Neg_LimitOutterRight;
    arAxisCtrl_gb[AxisNo.Allocate_X].SetupMode.FastVelo := CurrentData.Axes.Allocate_X.Homing.FastVelo;
    arAxisCtrl_gb[AxisNo.Allocate_X].SetupMode.SlowVelo := CurrentData.Axes.Allocate_X.Homing.SlowVelo;
    arAxisCtrl_gb[AxisNo.Allocate_X].SetupMode.lrOffset := CurrentData.Axes.Allocate_X.Homing.Offset;
    arAxisCtrl_gb[AxisNo.Allocate_X].SetupMode.lrSetPosition := CurrentData.Axes.Allocate_X.Homing.SetAbsolutePosition;
    arAxisCtrl_gb[AxisNo.Allocate_X].SetupMode.stPosBiasParameter.bSetPostionBias := TRUE;
    arAxisCtrl_gb[AxisNo.Allocate_X].Admin._OpMode.en := ModeHoming;
ELSIF TableMove.xBusy AND AllowAllocateRobotMove THEN
    arAxisCtrl_gb[AxisNo.Allocate_X].Admin._OpMode.en := ModePosAbs;
ELSIF fbAllocateArea.fbAllocateRobotNeedlingMove.xBusy AND AllowAllocateRobotMove THEN
	arAxisCtrl_gb[AxisNo.Allocate_X].PosMode.Acc := CurrentData.Axes.Allocate_X.Manual.PtpAcceleration;
    arAxisCtrl_gb[AxisNo.Allocate_X].PosMode.Dec := CurrentData.Axes.Allocate_X.Manual.PtpDeceleration;
    arAxisCtrl_gb[AxisNo.Allocate_X].PosMode.Jerk := CurrentData.Axes.Allocate_X.Manual.PtpJerk;
    arAxisCtrl_gb[AxisNo.Allocate_X].PosMode.Velocity := CurrentData.Axes.Allocate_X.Manual.PtpVelocity;
    arAxisCtrl_gb[AxisNo.Allocate_X].Admin._OpMode.en := ModePosAbs;	
  
ELSIF fbAllocateArea.fb_AllocateBatchMode.Busy AND AllowAllocateRobotMove THEN
    arAxisCtrl_gb[AxisNo.Allocate_X].Admin._OpMode.en := ModePosAbs;

					  
ELSE
    arAxisCtrl_gb[AxisNo.Allocate_X].Admin.StopDeceleration := 1000;
    arAxisCtrl_gb[AxisNo.Allocate_X].Admin._OpMode.en := E_AXIS_MODE.ModeAH;
		 
			 
END_IF
{endregion}

{region "AllocateRobot AxisY"}
IF AllocateManualCommand.AllocatedRobot.AxisY.JOG.MoveFWD AND AllowAllocateRobotMove THEN
    arAxisCtrl_gb[AxisNo.Allocate_Y].VelMode.Acc := CurrentData.Axes.Allocate_Y.Manual.JogAcceleration;
    arAxisCtrl_gb[AxisNo.Allocate_Y].VelMode.Dec := CurrentData.Axes.Allocate_Y.Manual.JogDeceleration;
    arAxisCtrl_gb[AxisNo.Allocate_Y].VelMode.Jerk := CurrentData.Axes.Allocate_Y.Manual.JogJerk;
    arAxisCtrl_gb[AxisNo.Allocate_Y].VelMode.Velocity := CurrentData.Axes.Allocate_Y.Manual.JogVelocity;
    arAxisCtrl_gb[AxisNo.Allocate_Y].Admin._OpMode.en := E_AXIS_MODE.ModeVel;
ELSIF AllocateManualCommand.AllocatedRobot.AxisY.JOG.MoveBWD AND AllowAllocateRobotMove THEN
    arAxisCtrl_gb[AxisNo.Allocate_Y].VelMode.Acc := CurrentData.Axes.Allocate_Y.Manual.JogAcceleration;
    arAxisCtrl_gb[AxisNo.Allocate_Y].VelMode.Dec := CurrentData.Axes.Allocate_Y.Manual.JogDeceleration;
    arAxisCtrl_gb[AxisNo.Allocate_Y].VelMode.Jerk := CurrentData.Axes.Allocate_Y.Manual.JogJerk;
    arAxisCtrl_gb[AxisNo.Allocate_Y].VelMode.Velocity := CurrentData.Axes.Allocate_Y.Manual.JogVelocity * -1;
    arAxisCtrl_gb[AxisNo.Allocate_Y].Admin._OpMode.en := E_AXIS_MODE.ModeVel;
ELSIF AllocateManualCommand.AllocatedRobot.AxisY.PTP.Enable  AND AllowAllocateRobotMove THEN
    arAxisCtrl_gb[AxisNo.Allocate_Y].PosMode.Acc := CurrentData.Axes.Allocate_Y.Manual.PtpAcceleration;
    arAxisCtrl_gb[AxisNo.Allocate_Y].PosMode.Dec := CurrentData.Axes.Allocate_Y.Manual.PtpDeceleration;
    arAxisCtrl_gb[AxisNo.Allocate_Y].PosMode.Jerk := CurrentData.Axes.Allocate_Y.Manual.PtpJerk;
    arAxisCtrl_gb[AxisNo.Allocate_Y].PosMode.Velocity := CurrentData.Axes.Allocate_Y.Manual.PtpVelocity;
    arAxisCtrl_gb[AxisNo.Allocate_Y].PosMode.Position := CurrentData.Axes.Allocate_Y.Manual.PtpPosition;
    arAxisCtrl_gb[AxisNo.Allocate_Y].Admin._OpMode.en := ModePosAbs;
//ELSIF( AllocateManualCommand.AllocatedRobot.AxisY.Homing.Execute OR  fbAllocateArea.fbAllocateHome.AxisHomingRequest ) AND AllowAllocateRobotMove THEN
//    arAxisCtrl_gb[AxisNo.Allocate_Y].SetupMode.eHomingMode := E_HomingMode._36_MoveToAbsHomePoint;
//    arAxisCtrl_gb[AxisNo.Allocate_Y].SetupMode.FastVelo := CurrentData.Axes.Allocate_Y.Homing.FastVelo;
//    arAxisCtrl_gb[AxisNo.Allocate_Y].SetupMode.SlowVelo := CurrentData.Axes.Allocate_Y.Homing.SlowVelo;
//    arAxisCtrl_gb[AxisNo.Allocate_Y].SetupMode.lrOffset := CurrentData.Axes.Allocate_Y.Homing.Offset;
//    arAxisCtrl_gb[AxisNo.Allocate_Y].SetupMode.lrSetPosition := CurrentData.Axes.Allocate_Y.Homing.SetAbsolutePosition;
//    arAxisCtrl_gb[AxisNo.Allocate_Y].SetupMode.stPosBiasParameter.bSetPostionBias := FALSE;
//    arAxisCtrl_gb[AxisNo.Allocate_Y].Admin._OpMode.en := ModeHoming;
ELSIF( AllocateManualCommand.AllocatedRobot.AxisY.Homing.Execute OR  fbAllocateArea.fbAllocateHome.AxisHomingRequest ) AND AllowAllocateRobotMove THEN
	GVL_Machine.AllocatYAxisHome := FALSE;
    arAxisCtrl_gb[AxisNo.Allocate_Y].PosMode.Acc := CurrentData.Axes.Allocate_Y.Homing.FastVelo.Acc;
    arAxisCtrl_gb[AxisNo.Allocate_Y].PosMode.Dec := CurrentData.Axes.Allocate_Y.Homing.FastVelo.Dec;
    arAxisCtrl_gb[AxisNo.Allocate_Y].PosMode.Jerk := CurrentData.Axes.Allocate_Y.Homing.FastVelo.Jerk;
    arAxisCtrl_gb[AxisNo.Allocate_Y].PosMode.Velocity := CurrentData.Axes.Allocate_Y.Homing.FastVelo.Velocity;
    arAxisCtrl_gb[AxisNo.Allocate_Y].PosMode.Position := CurrentData.Axes.Allocate_Y.Homing.Offset;
    arAxisCtrl_gb[AxisNo.Allocate_Y].Admin._OpMode.en := ModePosAbs;
		 
    IF arAxisStatus_gb[AxisNo.Allocate_Y].Admin._OpModeAck = ModePosAbs AND arAxisStatus_gb[AxisNo.Allocate_Y].Admin.CmdDone THEN
        GVL_Machine.AllocatYAxisHome := TRUE;
    END_IF
ELSIF TableMove.xBusy AND AllowAllocateRobotMove THEN
    arAxisCtrl_gb[AxisNo.Allocate_Y].Admin._OpMode.en := ModePosAbs;
ELSIF fbAllocateArea.fb_AllocateBatchMode.Busy AND AllowAllocateRobotMove THEN
    arAxisCtrl_gb[AxisNo.Allocate_Y].Admin._OpMode.en := ModePosAbs;
ELSIF fbAllocateArea.fbAllocateRobotNeedlingMove.xBusy AND AllowAllocateRobotMove THEN
	arAxisCtrl_gb[AxisNo.Allocate_Y].PosMode.Acc := CurrentData.Axes.Allocate_Y.Manual.PtpAcceleration;
    arAxisCtrl_gb[AxisNo.Allocate_Y].PosMode.Dec := CurrentData.Axes.Allocate_Y.Manual.PtpDeceleration;
    arAxisCtrl_gb[AxisNo.Allocate_Y].PosMode.Jerk := CurrentData.Axes.Allocate_Y.Manual.PtpJerk;
    arAxisCtrl_gb[AxisNo.Allocate_Y].PosMode.Velocity := CurrentData.Axes.Allocate_Y.Manual.PtpVelocity;
    arAxisCtrl_gb[AxisNo.Allocate_Y].Admin._OpMode.en := ModePosAbs;
ELSE
    arAxisCtrl_gb[AxisNo.Allocate_Y].Admin.StopDeceleration := 1000;
    arAxisCtrl_gb[AxisNo.Allocate_Y].Admin._OpMode.en := E_AXIS_MODE.ModeAH;
END_IF

{EndRegion}

{region "OutRobot AxisX"}
IF AllocateManualCommand.OutRobot.AxisX.JOG.MoveFWD AND AllowOutRobotMove THEN
    arAxisCtrl_gb[AxisNo.OutRobot_X].VelMode.Acc := CurrentData.Axes.OutRobot_X.Manual.JogAcceleration;
    arAxisCtrl_gb[AxisNo.OutRobot_X].VelMode.Dec := CurrentData.Axes.OutRobot_X.Manual.JogDeceleration;
    arAxisCtrl_gb[AxisNo.OutRobot_X].VelMode.Jerk := CurrentData.Axes.OutRobot_X.Manual.JogJerk;
    arAxisCtrl_gb[AxisNo.OutRobot_X].VelMode.Velocity := CurrentData.Axes.OutRobot_X.Manual.JogVelocity;
    arAxisCtrl_gb[AxisNo.OutRobot_X].Admin._OpMode.en := E_AXIS_MODE.ModeVel;
ELSIF AllocateManualCommand.OutRobot.AxisX.JOG.MoveBWD AND AllowOutRobotMove THEN
    arAxisCtrl_gb[AxisNo.OutRobot_X].VelMode.Acc := CurrentData.Axes.OutRobot_X.Manual.JogAcceleration;
    arAxisCtrl_gb[AxisNo.OutRobot_X].VelMode.Dec := CurrentData.Axes.OutRobot_X.Manual.JogDeceleration;
    arAxisCtrl_gb[AxisNo.OutRobot_X].VelMode.Jerk := CurrentData.Axes.OutRobot_X.Manual.JogJerk;
    arAxisCtrl_gb[AxisNo.OutRobot_X].VelMode.Velocity := CurrentData.Axes.OutRobot_X.Manual.JogVelocity * -1;
    arAxisCtrl_gb[AxisNo.OutRobot_X].Admin._OpMode.en := E_AXIS_MODE.ModeVel;
ELSIF AllocateManualCommand.OutRobot.AxisX.PTP.Enable AND AllowOutRobotMove THEN
    arAxisCtrl_gb[AxisNo.OutRobot_X].PosMode.Acc := CurrentData.Axes.OutRobot_X.Manual.PtpAcceleration;
    arAxisCtrl_gb[AxisNo.OutRobot_X].PosMode.Dec := CurrentData.Axes.OutRobot_X.Manual.PtpDeceleration;
    arAxisCtrl_gb[AxisNo.OutRobot_X].PosMode.Jerk := CurrentData.Axes.OutRobot_X.Manual.PtpJerk;
    arAxisCtrl_gb[AxisNo.OutRobot_X].PosMode.Velocity := CurrentData.Axes.OutRobot_X.Manual.PtpVelocity;
    arAxisCtrl_gb[AxisNo.OutRobot_X].PosMode.Position := CurrentData.Axes.OutRobot_X.Manual.PtpPosition;
    arAxisCtrl_gb[AxisNo.OutRobot_X].Admin._OpMode.en := ModePosAbs;
ELSIF (AllocateManualCommand.OutRobot.AxisX.Homing.Execute OR  fbAllocateArea.fbAllocateHome.AxisHomingRequest ) AND AllowOutRobotMove THEN
    arAxisCtrl_gb[AxisNo.OutRobot_X].SetupMode.eHomingMode := E_HomingMode._28_Neg_HomeInnerRight_withLimit;
    arAxisCtrl_gb[AxisNo.OutRobot_X].SetupMode.FastVelo := CurrentData.Axes.OutRobot_X.Homing.FastVelo;
    arAxisCtrl_gb[AxisNo.OutRobot_X].SetupMode.SlowVelo := CurrentData.Axes.OutRobot_X.Homing.SlowVelo;
    arAxisCtrl_gb[AxisNo.OutRobot_X].SetupMode.lrOffset := CurrentData.Axes.OutRobot_X.Homing.Offset;
    arAxisCtrl_gb[AxisNo.OutRobot_X].SetupMode.lrSetPosition := CurrentData.Axes.OutRobot_X.Homing.SetAbsolutePosition;
    arAxisCtrl_gb[AxisNo.OutRobot_X].SetupMode.stPosBiasParameter.bSetPostionBias := TRUE;
    arAxisCtrl_gb[AxisNo.OutRobot_X].Admin._OpMode.en := ModeHoming;
ELSIF TableMove.xBusy AND AllowOutRobotMove THEN
	arAxisCtrl_gb[AxisNo.OutRobot_X].Admin._OpMode.en := ModePosAbs;
ELSIF (AllocateService.AutoMode_BoxMoveReverse.HandShake.Busy 
	  OR AllocateService.AutoMode_EmptyBoxMove.HandShake.Busy 
	  OR AllocateService.AutoMode_RareBoxMove.HandShake.Busy) AND AllowOutRobotMove THEN
	arAxisCtrl_gb[AxisNo.OutRobot_X].PosMode.Acc := CurrentData.Axes.OutRobot_X.HalfAuto.Acceleration;
    arAxisCtrl_gb[AxisNo.OutRobot_X].PosMode.Dec := CurrentData.Axes.OutRobot_X.HalfAuto.Deceleration;
    arAxisCtrl_gb[AxisNo.OutRobot_X].PosMode.Jerk := CurrentData.Axes.OutRobot_X.HalfAuto.Jerk;
    arAxisCtrl_gb[AxisNo.OutRobot_X].PosMode.Velocity := CurrentData.Axes.OutRobot_X.HalfAuto.Velocity;		   
    arAxisCtrl_gb[AxisNo.OutRobot_X].Admin._OpMode.en := ModePosAbs;
ELSE
    arAxisCtrl_gb[AxisNo.OutRobot_X].Admin.StopDeceleration := 1000;
    arAxisCtrl_gb[AxisNo.OutRobot_X].Admin._OpMode.en := E_AXIS_MODE.ModeAH;
END_IF

{Endregion}

{region "OutRobot AxisY"}
IF AllocateManualCommand.OutRobot.AxisY.JOG.MoveFWD AND AllowOutRobotMove THEN
    arAxisCtrl_gb[AxisNo.OutRobot_Y].VelMode.Acc := CurrentData.Axes.OutRobot_Y.Manual.JogAcceleration;
    arAxisCtrl_gb[AxisNo.OutRobot_Y].VelMode.Dec := CurrentData.Axes.OutRobot_Y.Manual.JogDeceleration;
    arAxisCtrl_gb[AxisNo.OutRobot_Y].VelMode.Jerk := CurrentData.Axes.OutRobot_Y.Manual.JogJerk;
    arAxisCtrl_gb[AxisNo.OutRobot_Y].VelMode.Velocity := CurrentData.Axes.OutRobot_Y.Manual.JogVelocity;
    arAxisCtrl_gb[AxisNo.OutRobot_Y].Admin._OpMode.en := E_AXIS_MODE.ModeVel;
ELSIF AllocateManualCommand.OutRobot.AxisY.JOG.MoveBWD AND AllowOutRobotMove THEN
    arAxisCtrl_gb[AxisNo.OutRobot_Y].VelMode.Acc := CurrentData.Axes.OutRobot_Y.Manual.JogAcceleration;
    arAxisCtrl_gb[AxisNo.OutRobot_Y].VelMode.Dec := CurrentData.Axes.OutRobot_Y.Manual.JogDeceleration;
    arAxisCtrl_gb[AxisNo.OutRobot_Y].VelMode.Jerk := CurrentData.Axes.OutRobot_Y.Manual.JogJerk;
    arAxisCtrl_gb[AxisNo.OutRobot_Y].VelMode.Velocity := CurrentData.Axes.OutRobot_Y.Manual.JogVelocity * -1;
    arAxisCtrl_gb[AxisNo.OutRobot_Y].Admin._OpMode.en := E_AXIS_MODE.ModeVel;
ELSIF AllocateManualCommand.OutRobot.AxisY.PTP.Enable AND AllowOutRobotMove THEN
    arAxisCtrl_gb[AxisNo.OutRobot_Y].PosMode.Acc := CurrentData.Axes.OutRobot_Y.Manual.PtpAcceleration;
    arAxisCtrl_gb[AxisNo.OutRobot_Y].PosMode.Dec := CurrentData.Axes.OutRobot_Y.Manual.PtpDeceleration;
    arAxisCtrl_gb[AxisNo.OutRobot_Y].PosMode.Jerk := CurrentData.Axes.OutRobot_Y.Manual.PtpJerk;
    arAxisCtrl_gb[AxisNo.OutRobot_Y].PosMode.Velocity := CurrentData.Axes.OutRobot_Y.Manual.PtpVelocity;
    arAxisCtrl_gb[AxisNo.OutRobot_Y].PosMode.Position := CurrentData.Axes.OutRobot_Y.Manual.PtpPosition;
    arAxisCtrl_gb[AxisNo.OutRobot_Y].Admin._OpMode.en := ModePosAbs;
ELSIF (AllocateManualCommand.OutRobot.AxisY.Homing.Execute OR  fbAllocateArea.fbAllocateHome.AxisHomingRequest) AND AllowOutRobotMove THEN
    arAxisCtrl_gb[AxisNo.OutRobot_Y].SetupMode.eHomingMode := E_HomingMode._28_Neg_HomeInnerRight_withLimit;
    arAxisCtrl_gb[AxisNo.OutRobot_Y].SetupMode.FastVelo := CurrentData.Axes.OutRobot_Y.Homing.FastVelo;
    arAxisCtrl_gb[AxisNo.OutRobot_Y].SetupMode.SlowVelo := CurrentData.Axes.OutRobot_Y.Homing.SlowVelo;
    arAxisCtrl_gb[AxisNo.OutRobot_Y].SetupMode.lrOffset := CurrentData.Axes.OutRobot_Y.Homing.Offset;
    arAxisCtrl_gb[AxisNo.OutRobot_Y].SetupMode.lrSetPosition := CurrentData.Axes.OutRobot_Y.Homing.SetAbsolutePosition;
    arAxisCtrl_gb[AxisNo.OutRobot_Y].SetupMode.stPosBiasParameter.bSetPostionBias := TRUE;
    arAxisCtrl_gb[AxisNo.OutRobot_Y].Admin._OpMode.en := ModeHoming;
ELSIF TableMove.xBusy AND AllowOutRobotMove THEN
	arAxisCtrl_gb[AxisNo.OutRobot_Y].Admin._OpMode.en := ModePosAbs;
ELSIF (AllocateService.AutoMode_BoxMoveReverse.HandShake.Busy 
	  OR AllocateService.AutoMode_EmptyBoxMove.HandShake.Busy 
	  OR AllocateService.AutoMode_RareBoxMove.HandShake.Busy)AND AllowOutRobotMove THEN
	arAxisCtrl_gb[AxisNo.OutRobot_Y].PosMode.Acc := CurrentData.Axes.OutRobot_Y.HalfAuto.Acceleration;
    arAxisCtrl_gb[AxisNo.OutRobot_Y].PosMode.Dec := CurrentData.Axes.OutRobot_Y.HalfAuto.Deceleration;
    arAxisCtrl_gb[AxisNo.OutRobot_Y].PosMode.Jerk := CurrentData.Axes.OutRobot_Y.HalfAuto.Jerk;
    arAxisCtrl_gb[AxisNo.OutRobot_Y].PosMode.Velocity := CurrentData.Axes.OutRobot_Y.HalfAuto.Velocity;		   
    arAxisCtrl_gb[AxisNo.OutRobot_Y].Admin._OpMode.en := ModePosAbs;
ELSE
    arAxisCtrl_gb[AxisNo.OutRobot_Y].Admin.StopDeceleration := 1000;
    arAxisCtrl_gb[AxisNo.OutRobot_Y].Admin._OpMode.en := E_AXIS_MODE.ModeAH;
END_IF

{Endregion}

{region "RoundBelt Axis"}
IF AllocateManualCommand.RoundBelt.Axis.JOG.MoveFWD AND AllowRoundBeltMove THEN
    arAxisCtrl_gb[AxisNo.RoundBelt].VelMode.Acc := CurrentData.Axes.RoundBelt.Manual.JogAcceleration;
    arAxisCtrl_gb[AxisNo.RoundBelt].VelMode.Dec := CurrentData.Axes.RoundBelt.Manual.JogDeceleration;
    arAxisCtrl_gb[AxisNo.RoundBelt].VelMode.Jerk := CurrentData.Axes.RoundBelt.Manual.JogJerk;
    arAxisCtrl_gb[AxisNo.RoundBelt].VelMode.Velocity := CurrentData.Axes.RoundBelt.Manual.JogVelocity;
    arAxisCtrl_gb[AxisNo.RoundBelt].Admin._OpMode.en := E_AXIS_MODE.ModeVel;
ELSIF AllocateManualCommand.RoundBelt.Axis.JOG.MoveBWD AND AllowRoundBeltMove THEN
    arAxisCtrl_gb[AxisNo.RoundBelt].VelMode.Acc := CurrentData.Axes.RoundBelt.Manual.JogAcceleration;
    arAxisCtrl_gb[AxisNo.RoundBelt].VelMode.Dec := CurrentData.Axes.RoundBelt.Manual.JogDeceleration;
    arAxisCtrl_gb[AxisNo.RoundBelt].VelMode.Jerk := CurrentData.Axes.RoundBelt.Manual.JogJerk;
    arAxisCtrl_gb[AxisNo.RoundBelt].VelMode.Velocity := CurrentData.Axes.RoundBelt.Manual.JogVelocity * -1;
    arAxisCtrl_gb[AxisNo.RoundBelt].Admin._OpMode.en := E_AXIS_MODE.ModeVel;
ELSIF AllocateManualCommand.RoundBelt.Axis.PTP.Enable AND AllowRoundBeltMove THEN
    arAxisCtrl_gb[AxisNo.RoundBelt].PosMode.Acc := CurrentData.Axes.RoundBelt.Manual.PtpAcceleration;
    arAxisCtrl_gb[AxisNo.RoundBelt].PosMode.Dec := CurrentData.Axes.RoundBelt.Manual.PtpDeceleration;
    arAxisCtrl_gb[AxisNo.RoundBelt].PosMode.Jerk := CurrentData.Axes.RoundBelt.Manual.PtpJerk;
    arAxisCtrl_gb[AxisNo.RoundBelt].PosMode.Velocity := CurrentData.Axes.RoundBelt.Manual.PtpVelocity;
    arAxisCtrl_gb[AxisNo.RoundBelt].PosMode.Position := CurrentData.Axes.RoundBelt.Manual.PtpPosition;
    arAxisCtrl_gb[AxisNo.RoundBelt].Admin._OpMode.en := ModePosAbs;
ELSIF (AllocateManualCommand.RoundBelt.Axis.Homing.Execute OR  fbAllocateArea.fbAllocateHome.AxisHomingRequest ) AND AllowRoundBeltMove THEN
    arAxisCtrl_gb[AxisNo.RoundBelt].SetupMode.eHomingMode := E_HomingMode._20_Pos_HomeInnerLeft;
    arAxisCtrl_gb[AxisNo.RoundBelt].SetupMode.FastVelo := CurrentData.Axes.RoundBelt.Homing.FastVelo;
    arAxisCtrl_gb[AxisNo.RoundBelt].SetupMode.SlowVelo := CurrentData.Axes.RoundBelt.Homing.SlowVelo;
    arAxisCtrl_gb[AxisNo.RoundBelt].SetupMode.lrOffset := CurrentData.Axes.RoundBelt.Homing.Offset;
    arAxisCtrl_gb[AxisNo.RoundBelt].SetupMode.lrSetPosition := CurrentData.Axes.RoundBelt.Homing.SetAbsolutePosition;
    arAxisCtrl_gb[AxisNo.RoundBelt].SetupMode.stPosBiasParameter.bSetPostionBias := TRUE;
    arAxisCtrl_gb[AxisNo.RoundBelt].Admin._OpMode.en := ModeHoming;
ELSIF TableMove.xBusy AND AllowRoundBeltMove THEN
    arAxisCtrl_gb[AxisNo.RoundBelt].Admin._OpMode.en := ModePosAbs;
ELSIF AllocateService.AllocateCircleMove.HandShake.Busy AND AllowRoundBeltMove THEN
    arAxisCtrl_gb[AxisNo.RoundBelt].PosMode.Acc := CurrentData.Axes.RoundBelt.HalfAuto.Acceleration;
    arAxisCtrl_gb[AxisNo.RoundBelt].PosMode.Dec := CurrentData.Axes.RoundBelt.HalfAuto.Deceleration;
    arAxisCtrl_gb[AxisNo.RoundBelt].PosMode.Jerk := CurrentData.Axes.RoundBelt.HalfAuto.Jerk;
    arAxisCtrl_gb[AxisNo.RoundBelt].PosMode.Velocity := CurrentData.Axes.RoundBelt.HalfAuto.Velocity;
    arAxisCtrl_gb[AxisNo.RoundBelt].Admin._OpMode.en := ModePosAbs;
ELSIF (AllocateService.AutoMode_AllocateBatchMode.HandShake.Busy OR StorageService.AutoMode_ReloadRoundBeltBoxWithRobot.Status.Busy) AND AllowRoundBeltMove THEN
    arAxisCtrl_gb[AxisNo.RoundBelt].PosMode.Acc := CurrentData.Axes.RoundBelt.HalfAuto.Acceleration;
    arAxisCtrl_gb[AxisNo.RoundBelt].PosMode.Dec := CurrentData.Axes.RoundBelt.HalfAuto.Deceleration;
    arAxisCtrl_gb[AxisNo.RoundBelt].PosMode.Jerk := CurrentData.Axes.RoundBelt.HalfAuto.Jerk;
    arAxisCtrl_gb[AxisNo.RoundBelt].PosMode.Velocity := CurrentData.Axes.RoundBelt.HalfAuto.Velocity;
    arAxisCtrl_gb[AxisNo.RoundBelt].Admin._OpMode.en := ModePosAbs;
ELSE
    arAxisCtrl_gb[AxisNo.RoundBelt].Admin.StopDeceleration := 1000;
    arAxisCtrl_gb[AxisNo.RoundBelt].Admin._OpMode.en := E_AXIS_MODE.ModeAH;
END_IF

{endregion}

{region "TurnTable Axis"}
IF AllocateManualCommand.TurnTable.Axis.JOG.MoveFWD AND AllowTurnTable THEN
    arAxisCtrl_gb[AxisNo.TurnTable].VelMode.Acc := CurrentData.Axes.TurnTable.Manual.JogAcceleration;
    arAxisCtrl_gb[AxisNo.TurnTable].VelMode.Dec := CurrentData.Axes.TurnTable.Manual.JogDeceleration;
    arAxisCtrl_gb[AxisNo.TurnTable].VelMode.Jerk := CurrentData.Axes.TurnTable.Manual.JogJerk;
    arAxisCtrl_gb[AxisNo.TurnTable].VelMode.Velocity := CurrentData.Axes.TurnTable.Manual.JogVelocity;
    arAxisCtrl_gb[AxisNo.TurnTable].Admin._OpMode.en := E_AXIS_MODE.ModeVel;
ELSIF AllocateManualCommand.TurnTable.Axis.JOG.MoveBWD THEN
    arAxisCtrl_gb[AxisNo.TurnTable].VelMode.Acc := CurrentData.Axes.TurnTable.Manual.JogAcceleration;
    arAxisCtrl_gb[AxisNo.TurnTable].VelMode.Dec := CurrentData.Axes.TurnTable.Manual.JogDeceleration;
    arAxisCtrl_gb[AxisNo.TurnTable].VelMode.Jerk := CurrentData.Axes.TurnTable.Manual.JogJerk;
    arAxisCtrl_gb[AxisNo.TurnTable].VelMode.Velocity := CurrentData.Axes.TurnTable.Manual.JogVelocity * -1;
    arAxisCtrl_gb[AxisNo.TurnTable].Admin._OpMode.en := E_AXIS_MODE.ModeVel;
ELSIF AllocateManualCommand.TurnTable.Axis.PTP.Enable THEN
    arAxisCtrl_gb[AxisNo.TurnTable].PosMode.Acc := CurrentData.Axes.TurnTable.Manual.PtpAcceleration;
    arAxisCtrl_gb[AxisNo.TurnTable].PosMode.Dec := CurrentData.Axes.TurnTable.Manual.PtpDeceleration;
    arAxisCtrl_gb[AxisNo.TurnTable].PosMode.Jerk := CurrentData.Axes.TurnTable.Manual.PtpJerk;
    arAxisCtrl_gb[AxisNo.TurnTable].PosMode.Velocity := CurrentData.Axes.TurnTable.Manual.PtpVelocity;
    arAxisCtrl_gb[AxisNo.TurnTable].PosMode.Position := CurrentData.Axes.TurnTable.Manual.PtpPosition;
    arAxisCtrl_gb[AxisNo.TurnTable].Admin._OpMode.en := ModePosAbs;
ELSIF (AllocateManualCommand.TurnTable.Axis.Homing.Execute OR  fbAllocateArea.fbAllocateHome.AxisHomingRequest) AND  AllowTurnTable THEN
    arAxisCtrl_gb[AxisNo.TurnTable].SetupMode.eHomingMode := E_HomingMode._22_Neg_HomeInnerRight;
    arAxisCtrl_gb[AxisNo.TurnTable].SetupMode.FastVelo := CurrentData.Axes.TurnTable.Homing.FastVelo;
    arAxisCtrl_gb[AxisNo.TurnTable].SetupMode.SlowVelo := CurrentData.Axes.TurnTable.Homing.SlowVelo;
    arAxisCtrl_gb[AxisNo.TurnTable].SetupMode.lrOffset := CurrentData.Axes.TurnTable.Homing.Offset;
    arAxisCtrl_gb[AxisNo.TurnTable].SetupMode.lrSetPosition := CurrentData.Axes.TurnTable.Homing.SetAbsolutePosition;
    arAxisCtrl_gb[AxisNo.TurnTable].SetupMode.stPosBiasParameter.bSetPostionBias := TRUE;
    arAxisCtrl_gb[AxisNo.TurnTable].Admin._OpMode.en := ModeHoming;
ELSIF TableMove.xBusy AND AllowTurnTable THEN
    arAxisCtrl_gb[AxisNo.TurnTable].Admin._OpMode.en := ModePosAbs;
ELSIF AllocateService.TurnTableMove.HandShake.Busy AND AllowTurnTable THEN
    arAxisCtrl_gb[AxisNo.TurnTable].PosMode.Acc := CurrentData.Axes.TurnTable.HalfAuto.Acceleration;
    arAxisCtrl_gb[AxisNo.TurnTable].PosMode.Dec := CurrentData.Axes.TurnTable.HalfAuto.Deceleration;
    arAxisCtrl_gb[AxisNo.TurnTable].PosMode.Jerk := CurrentData.Axes.TurnTable.HalfAuto.Jerk;
    arAxisCtrl_gb[AxisNo.TurnTable].PosMode.Velocity := CurrentData.Axes.TurnTable.HalfAuto.Velocity;
    arAxisCtrl_gb[AxisNo.TurnTable].Admin._OpMode.en := ModePosAbs;
ELSE
    arAxisCtrl_gb[AxisNo.TurnTable].Admin.StopDeceleration := 1000;
    arAxisCtrl_gb[AxisNo.TurnTable].Admin._OpMode.en := E_AXIS_MODE.ModeAH;
END_IF

{endregion}

{region "Rack motor Axis"}
IF StorageManualCommand.RackMotor.Axis.JOG.MoveFWD AND AllowRackMotor THEN
    arAxisCtrl_gb[AxisNo.RackMotor].VelMode.Acc := CurrentData.Axes.RackMotor.Manual.JogAcceleration;
    arAxisCtrl_gb[AxisNo.RackMotor].VelMode.Dec := CurrentData.Axes.RackMotor.Manual.JogDeceleration;
    arAxisCtrl_gb[AxisNo.RackMotor].VelMode.Jerk := CurrentData.Axes.RackMotor.Manual.JogJerk;
    arAxisCtrl_gb[AxisNo.RackMotor].VelMode.Velocity := CurrentData.Axes.RackMotor.Manual.JogVelocity;
    arAxisCtrl_gb[AxisNo.RackMotor].Admin._OpMode.en := E_AXIS_MODE.ModeVel;
ELSIF StorageManualCommand.RackMotor.Axis.JOG.MoveBWD AND AllowRackMotor THEN
    arAxisCtrl_gb[AxisNo.RackMotor].VelMode.Acc := CurrentData.Axes.RackMotor.Manual.JogAcceleration;
    arAxisCtrl_gb[AxisNo.RackMotor].VelMode.Dec := CurrentData.Axes.RackMotor.Manual.JogDeceleration;
    arAxisCtrl_gb[AxisNo.RackMotor].VelMode.Jerk := CurrentData.Axes.RackMotor.Manual.JogJerk;
    arAxisCtrl_gb[AxisNo.RackMotor].VelMode.Velocity := CurrentData.Axes.RackMotor.Manual.JogVelocity * -1;
    arAxisCtrl_gb[AxisNo.RackMotor].Admin._OpMode.en := E_AXIS_MODE.ModeVel;
ELSIF StorageManualCommand.RackMotor.Axis.PTP.Enable AND AllowRackMotor THEN
    arAxisCtrl_gb[AxisNo.RackMotor].PosMode.Acc := CurrentData.Axes.RackMotor.Manual.PtpAcceleration;
    arAxisCtrl_gb[AxisNo.RackMotor].PosMode.Dec := CurrentData.Axes.RackMotor.Manual.PtpDeceleration;
    arAxisCtrl_gb[AxisNo.RackMotor].PosMode.Jerk := CurrentData.Axes.RackMotor.Manual.PtpJerk;
    arAxisCtrl_gb[AxisNo.RackMotor].PosMode.Velocity := CurrentData.Axes.RackMotor.Manual.PtpVelocity;
    arAxisCtrl_gb[AxisNo.RackMotor].PosMode.Position := CurrentData.Axes.RackMotor.Manual.PtpPosition;
    arAxisCtrl_gb[AxisNo.RackMotor].Admin._OpMode.en := ModePosAbs;
ELSIF (StorageManualCommand.RackMotor.Axis.Homing.Execute OR fbStorageArea.fbStorageHoming.RackMotorHomeRequest) AND AllowRackMotor THEN
    arAxisCtrl_gb[AxisNo.RackMotor].SetupMode.eHomingMode := E_HomingMode._17_Neg_LimitOutterRight;
    arAxisCtrl_gb[AxisNo.RackMotor].SetupMode.FastVelo := CurrentData.Axes.RackMotor.Homing.FastVelo;
    arAxisCtrl_gb[AxisNo.RackMotor].SetupMode.SlowVelo := CurrentData.Axes.RackMotor.Homing.SlowVelo;
    arAxisCtrl_gb[AxisNo.RackMotor].SetupMode.lrOffset := CurrentData.Axes.RackMotor.Homing.Offset;
    arAxisCtrl_gb[AxisNo.RackMotor].SetupMode.lrSetPosition := CurrentData.Axes.RackMotor.Homing.SetAbsolutePosition;
    arAxisCtrl_gb[AxisNo.RackMotor].SetupMode.stPosBiasParameter.bSetPostionBias := TRUE;
    arAxisCtrl_gb[AxisNo.RackMotor].Admin._OpMode.en := ModeHoming;
ELSIF (TableMove.xBusy OR StorageService.AutoMode_AddBoxes.Status.Busy) AND AllowRackMotor THEN
    arAxisCtrl_gb[AxisNo.RackMotor].Admin._OpMode.en := ModePosAbs;
ELSIF fbStorageArea.fbBoxSupplyCtrl.Busy AND 
		fbStorageArea.fbBoxSupplyCtrl.AxisRackMotorBTNHomeRequest AND 
		AllowRackMotor THEN
	arAxisCtrl_gb[AxisNo.RackMotor].PosMode.Acc := CurrentData.Axes.RackMotor.HalfAuto.Acceleration;
	arAxisCtrl_gb[AxisNo.RackMotor].PosMode.Dec := CurrentData.Axes.RackMotor.HalfAuto.Deceleration;
	arAxisCtrl_gb[AxisNo.RackMotor].PosMode.Jerk := CurrentData.Axes.RackMotor.HalfAuto.Jerk;
	arAxisCtrl_gb[AxisNo.RackMotor].PosMode.Velocity := CurrentData.Axes.RackMotor.HalfAuto.Velocity;
	arAxisCtrl_gb[AxisNo.RackMotor].Admin._OpMode.en := ModePosAbs;
			 
ELSE
    arAxisCtrl_gb[AxisNo.RackMotor].Admin.StopDeceleration := 1000;
    arAxisCtrl_gb[AxisNo.RackMotor].Admin._OpMode.en := E_AXIS_MODE.ModeAH;
END_IF

{endregion}
END_METHOD

